# B&R Automation Studio project EFI (part 13)

#### Documentation.txt - Release Axis Ctrl Logic
```
 **************************************************************************************************
 * COPYRIGHT - B&R Spain
 **************************************************************************************************
 * Program: AxisCtrl
 * File: Documentation.txt
 * Author: B&R Spain
 * Created: September 19, 2013
 * Modified: April 28, 2017
 **************************************************************************************************
 * Implementation of program AxisCtrl
 **************************************************************************************************
 * V 0.03.4
 **************************************************************************************************

 * Requirements
 **************************************************************************************************

 - ACP10 version must be equal or higher than V2.26.0 because before that version the ACP10_MC FBK
   errors were not read by the MC_ReadAxisError FBK and therefore a lot of diagnostic information
   would be lost in case a previous version would be used.

 * Configuration
 **************************************************************************************************

 - The file References.st must be updated to allow the program to control the desired axis. This is
   the only part of the program that needs to be modified if the functionality does not need to be
   changed.

 - It must be noted that the name of the control variable is not used inside the program to avoid
   requiring a Find & Replace. The control variable just needs to be specified in the references.st
   file.

 * Functionality
 **************************************************************************************************

 - The funtionality is very similar to the SingleAx or Basic one. It basically has some expansions
   to allow higher flexibility. The interface is quite easy to use. Furthermore, there are some
   differences compared to the SingleAx and Basic programs, which are described in the following
   chapter.

 - The control structure is divided in three parts; the commands, the parameters and the status.

 - In addition to the PLCopen state, the control structure provides useful status information like
   the PowerOn, the HomeOk and the InPosition that reflects if the axis is switched on, if it is
   properly homed and if the last commanded discrete movement has reached the target, respectively.
   The status structure provides information about the ACOPOS digital inputs as well.

 * Main differences in behaviour compared to the SingleAx and Basic
 **************************************************************************************************

 - In this program, all the valid PLCopen transitions are possible. E.g. While a MoveAbsolute is
   performed (DiscreteMotion), a MoveVelocity can be started (ContinuousMotion). This includes as
   well performing a MoveAbsolute to a new target while a MoveAbsolute is in process. Not all the
   combinations were possible in the SingleAx and Basic programs.

 - Instead of a Stop, this program provides a Halt and a QuickStop.
   - The Halt allows Discrete, Continuous and synchronized movements to be halted (Discrete motion
     where the speed is decreased until it becomes zero). This allows a higher flexibility since
	 the Halt itself can be aborted by another movement or even a new Halt with other parameters.
	 This would be not possible if a Stop would be used.
   - The QuickStop performs a stop with the limit deceleration (Axis init table). The QuickStop can
     be thought of a "panic" stop. It has higher priority than any other command except switching
	 off the drive. If the QuickStop is set, no movement will be allowed to start. In case any un-
	 expected error occurrs, the QuickStop should be used to stop the motion.

 - The Quickstop and the Power must be reset by the application. This program will never reset them.

 - In this program, only the real axis errors (i.e. the ones that bring the axis to ErrorStop in
   the PLCopen state diagram. E.g. encoder fault) cause the axis to stop. If other errors (e.g.
   warnings or ACP10_MC errors (29xxx) occurr), the axis remains in its last state and can be ope-
   rated as normal. Therefore, the errors can be read (Acknowledged) while the axis is in motion.
   However, every error which is reported should be considered by the application and if necessary,
   command a QuikStop.

 - As the PLCopen state diagram states, the Reset command can be used to leave the ErrorStop state
   directly with no need to acknowledge the errors one by one. To mantain backwards compatibility,
   if all errors are acknowledged by the ErrorAcknowledge command, the axis leaves the ErrorStop
   state as well.

 - In this program, the homming mode cannot be specified by the application. Instead, there are
   three kind of home commands, which is enough for almost all applications.
   - The HomeDirect, which assigns a value to the actual position. This command can be used either
     in standstill or in disabled state.
   - The HomeAbsEncoder, which takes into account the absolute encoder to calculate the position.
     This command can be used either in standstill or in disabled state. To allow this functionality
	 a permanent variable must be linked, where the program will store the necessary data for it.
   - The Home, which performs a home in the way it is defined in the axis parameter table. this is
     the only home command that can cause the axis to move.

 - In this program, there are two kind of Jog commands; a continuous and an incremental one.

 - By default, if a command is set, which is not allowed at the time, the program returns an error.
   This behaviour can be changed by commenting the corresponding part of the program.

 - By default, if two or more incoherent commands are set at the same time, the axis ignores and
   resets all the commands (exept the QuickStop and the Power). This behaviour can be changed by
   commenting the corresponding part of the program.

 - This program has been designed to avoid all the known bugs from the SingleAx and Basic programs.

 - This program also fixes some ACP10 flaws. E.g. this program does not allow a periodic axis to be
   moved if it is not properly homed. This is not prevented by ACP10, and it might lead to very dan-
   gerous movements where the axis could collide against other machine parts.

 - There is a PLCopen state supervisor that makes sure that even if the axis is commanded by an ex-
   ternal source (e.g. the Test Window), it will always be possible to operate it from the program
   side (of course not while the Test is opened in Exclusive mode, but will work after it is closed).
   However, it is recommended not to move the axis from the Test Window, since the changes that it
   does are not monitored by PLCopen FBs. Moving the axis from the test window can cause the next
   movements to use speeds and accelerations other than the ones programmed.

 - The way the program gets access to the axes (ncaccess) makes sure that the program can be trans-
   fered in any mode (overload, copy or one cycle) and the program will still be able to manage the
   axis. No warm restart will be required, even after the first transfer.

 * Modifications: Recommended way to modify the program
 **************************************************************************************************

  In order to implement changes that require the use of a state machine, it is not always
  necessary to expand/modify the main sequence (AxisState state machine). Consider the possibility
  to use a new state machine specifically for that functionality. It will be much easier to
  implement and it will actually make more sense if it is not part of the main sequence. For
  instance, this would be the case of a manual brake operation, where the main sequence step does
  not need to be considered if the higher level application requires to set or release the brake.

  Depending on the changes to implement there are different strategies to follow:

  - If the program must be expanded but the main sequence is not going to be changed, for example
    in case the ActualTorque must be read, the program can be expanded just by doing as follows:

    1)  Modify the control structure AxisCtrl_typ or any derivative, and all necessary substructures.
    2)  Declare all needed FBKs instances and temporary variables.
    3)  Implement the FBK parameterization and call in the corresponding FBK call section in the
        AxisCtrl.st file.
    4)  Update the status values of the control structure in the last part of the AxisCtrl.st file.

  - In order to modify the main sequence in an appropiate way, next steps must be followed:

    1)  Modify the control structure AxisCtrl_typ or any derivative, and all necessary
        substructures.
    2)  Declare all needed FBKs instances and any temporary variable (AxisCtrl.var file). In case
        of movement FBKS, declare two instances ended in _0 and _1 to allow two consecutive motion
        commands of the same type.
    3)  Expand the AxisState_typ enumeration (AxisCtrl.typ file) to include the new required steps.
        In case of motion states, declare two states ended in _0 and _1 to allow two consecutive
        motion commands of the same type.
    4)  Define all the new necessary actions in the Commands.st file. In case of movement actions,
        declare two actions ended in _0 and _1 to allow two consecutive motion commands of the
        same type.
    5)  Add code to reset all the new commands in the ResetMotionCommands action (Commands.st).
    6)  Add code to reset all the new FBKs in the ResetExecutes action (Commands.st).
    7)  Implement the new steps in the CASE of the AxisCtrl.st file by following the same style
        used in the other steps.
    8)  Implement the FBK parameterization and call in the corresponding FBK call section in the
        AxisCtrl.st file.
    9)  Add the newly created steps in the CASE of the StateSupervisor.st considering in which
        PLCopen state the axis must be for each step, in order to detect any anomaly in the axis
        state.
    10) Add the possibility to perform the command (e.g. Move.CyclicPosition) wherever it should
        be possible (i.e. in every step of the CASE where it should be possible to do so) in the
	    AxisCtrl.st file. Keep the same style which is used in the other steps.
    11) In order to detect if any command is commanded when it connot be, add the corresponding
        code in the COMMAND INCOHERENCE CHECK section in the AxisCtrl.st file.
    12) In order to detect if two incoherent commands are commanded at the same time, add the
        corresponding code in the INVALID COMMAND ABORTION section in the AxisCtrl.st file.
    13) Update the status values of the control structure in the last part of the AxisCtrl.st file
        if necessary.
    14) Document all the important behavioural changes of the task in the Documentatioin.txt file.

 **************************************************************************************************
 * Revision History
 **************************************************************************************************
 * V0.03.4  2017-04-28
 * (change) Virtual axes exhibit now the same bahviour as real axes (PowerOn status corresponds to
 * the Power command and PLCopenState.Disabled and PLCopenState.Standstill status are consistent
 * to the Power command).
 * (change) The Power command is not set to TRUE by the program any more, because there is no need.
 * (bug fix) PowerOn status was set too early and that could incorrectly lead to error 29207
 * (bug fix) Some AR version (e.g. F4.03) do not copy the pointer's address when transferring in
 * copy mode. The program can work fine now with those AR versions as well.
 **************************************************************************************************
 * V0.03.3  2016-07-26
 * (Bug fix) The battery-backed (EBI) encoder errors were reset in more cases than strictly needed
 **************************************************************************************************
 * V0.03.2  2016-07-26
 * (new) Battery-backed (EBI) encoder errors can be directly acknowledged via the ErrorAcknowledge
 * command, for example during the first startup or after the encoder cable has been disconnected.
 * Internally, the task writes the ENCOD_COMMAND ParID to reset the econder error when necessary.
 * It must be noted that it is not possible to recover from a battery-backed (EBI) encoder error
 * via the Reset command. Only the ErrorAcknowledge command can recover the situation.
 * (new) If a battery-backed (EBI) encoder error is detected, the permanent memory that is used by
 * the mcHOME_RESTORE_POS is set to be invalid, because the absolute position could be wrong.
 * (Bug fix) Error message for MC_BR_AutControl was not correct
 **************************************************************************************************
 * V0.03.1  2016-02-17
 * (bug fix) If the axis lost the HomeOK due to an encoder error, the ActualPosition did not change
 * to NaN and the workaround introduced in V0.03.0 for the APC10 flaw was not preventing the axis
 * to move after an encoder error.
 * (bug fix) If the axis is not synchronized anymore due to an external abortion (e.g. because it
 * was stopped from the Test Window), the InGear and InSynch flag was not reset.
 * (change) Now the CommandAborted output from the different FBs is used to detect sooner if an
 * external agent (e.g the Test Window) is commanding other movements.
 * (change) If the program was transfered in overload mode while the axis state was not Standstill
 * or Disabled, the MC_BR_InitEndlessPosition was filling the error FIFO. Now it waits until it
 * can be executed and the InitDone remains FALSE until then.
 **************************************************************************************************
 * V0.03.0  2016-02-10
 * (change) If the axis is not properly referenced (HomeOK = FALSE), the ActualPosition shows Not
 * a Number (NaN) in order to avoid confusions.
 * (change) Error 50001 has been replaced by error 29207, which provides a more precise description
 * with detailed information about the FB which is responsible for it, making it easier to diagnose
 * application problems.
 * (new) If the axis is not properly referenced (HomeOK = FALSE), the axis is not allowed to
 * move by the application and error 29205 is reported. This is done because there is an ACP10 flaw
 * that allows rotary axes to move even if they are not homed and that could lead to dangerous
 * movements that might end colliding against some other machine part.
 * (new) The Status member ErrorSource has been added so that it is possible to know if the actual
 * error message has been reported by ACP10, by PLCopen or by the Task itself.
 * (new) The MC_BR_InitAutData has been added in the AutCtrl program to be able update the automat
 * parameters in a faster way after a second StartAutomat command.
 **************************************************************************************************
 * V0.02.9  2015-12-24
 * (new) The member PowerOn has been added to the Status structure so that it is possible to know
 * if power is supplied to the axis by just looking at it.
 **************************************************************************************************
 * V0.02.8  2015-05-06
 * (change) If the axis to control is a virtual axis, the Power command is automatically set to
 * TRUE by the program so that it will not cause PLCopen conflicts. This is because virtual axes
 * cannot be in Disabled state and the state supervisor would try to switch the axis off repeatedly
 * until the Power command would be set to TRUE.
 **************************************************************************************************
 * V0.02.7  2014-02-18
 * (new) There is a new sample (CamCtrl) to handle a cam profile coupling. Note that the Move.CamIn
 * command can only be used while the axis is not in SynchronizedMotion, so that to CamIn a second
 * time, first a CamOut or another aborting command must be commanded.
 * (new) There is a new sample (AutCtrl) to handle a cam profile automat coupling. Note that the
 * Move.StartAutomat command can be used while the axis is not in SynchronizedMotion to start the
 * automat, but can be commanded again to update the automat parameters during runtime.
 * (change) The GearOut did not work correctly.
 **************************************************************************************************
 * V0.02.6  2013-12-30
 * (change) The state supervisor has been changed so that if an exception is found, it takes into
 * account the actual state for every cicle, without waiting for any timeout. This was necessary
 * when the CNC/robotics was used, because the axis was changed to synchronized motion and back to
 * standstill by the CNC and then it was not possible to perform any movement before the timeout
 * expired.
 **************************************************************************************************
 * V0.02.5  2013-10-17
 * (new) There is a new sample (GearCtrl) to handle a gear coupling.
 * (change) The way to handle the FBK calls has changed to let the user know when the master axis
 * is not correct.
 **************************************************************************************************
 * V0.02.4  2013-09-30
 * (new) First internally released version.
 **************************************************************************************************
```

#### AxisCtrl.typ - Local data types
```iecst
(********************************************************************
 * COPYRIGHT - B&R Spain
 ********************************************************************
 * Program: AxisCtrl
 * File: AxisCtrl.typ
 * Author: B&R Spain
 * Created: September 19, 2013
 ********************************************************************
 * Local data types of program AxisCtrl
 ********************************************************************)

TYPE
	AxisState_typ :
		(
		AX_STATE_DISABLED := 0,
		AX_STATE_HOMING_NO_POWER := 1,
		AX_STATE_SWITCHING_OFF := 2,
		AX_STATE_STANDSTILL := 10,
		AX_STATE_SWITCHING_ON := 11,
		AX_STATE_STOPPING := 12,
		AX_STATE_HOMING := 13,
		AX_STATE_MOVING_ABSOLUTE_0 := 20,
		AX_STATE_MOVING_ABSOLUTE_1 := 21,
		AX_STATE_MOVING_ADDITIVE_0 := 22,
		AX_STATE_MOVING_ADDITIVE_1 := 23,
		AX_STATE_MOVING_VELOCITY_0 := 24,
		AX_STATE_MOVING_VELOCITY_1 := 25,
		AX_STATE_MOVING_GEAR_0 := 40,
		AX_STATE_MOVING_GEAR_1 := 41,
		AX_STATE_HALTING_0 := 26,
		AX_STATE_HALTING_1 := 27,
		AX_STATE_JOGGING_POS := 30,
		AX_STATE_JOGGING_NEG := 31,
		AX_STATE_JOGGING_SS_POS := 32,
		AX_STATE_JOGGING_SS_NEG := 33,
		AX_STATE_JOG_SS_HALTED := 34,
		AX_STATE_HALTING_JOG := 35,
		AX_STATE_UNKNOWN := 200,
		AX_STATE_UK_DISABLED := 201,
		AX_STATE_UK_STANDSTILL := 202,
		AX_STATE_UK_HOMING := 203,
		AX_STATE_UK_DISCRETE_MOTION := 204,
		AX_STATE_UK_CONTINUOUS_MOTION := 205,
		AX_STATE_UK_SYNCHRONIZED_MOTION := 206,
		AX_STATE_UK_STOPPING := 207,
		AX_STATE_UK_ERROR_STOP := 208
		);
	AxisErrorState_typ :
		(
		AX_ERR_STATE_WAIT := 100, (*constant for the waiting error step*)
		AX_ERR_STATE_APP_ERROR := 101, (*constant for the application error step*)
		AX_ERR_STATE_AXIS_ERROR := 102, (*constant for the axis error step*)
		AX_ERR_STATE_ENCODER_RESET := 103 (*constant for the step where the encoder error is reset*)
		);
END_TYPE
```

- Program Logical/ExtPack/_Motion/AxisCtrl/AxisCtrl_v2/InitAxisControl (IEC) - Init Axis Control Index (no source held here)

### AxisCtrlGen.var - Global Axis Vars
```iecst
VAR
	gIndexAxisCtrl : INT := 1; (* Initialize Index*)
END_VAR
```

### Icla.typ
```iecst
(*********************************************************************************
 * Copyright: Bernecker + Rainer
 * Author:    gimeneza
 * Created:   June 15, 2017/4:14 PM
 *********************************************************************************)

TYPE
	stIcla_Error : 	STRUCT
		Jog : BOOL;
		Communication : BOOL;
		ErrorNumber : UINT;
	END_STRUCT;
	stIcla_Jog : 	STRUCT
		VeloSlow : UINT := 300; (*Rev/min Limited from 300 to 5000. 300 is the default value in Icla*)
		VeloFast : UINT := 1000; (*Rev/min Limited from 300 to 5000. 1000 is the default value in Icla*)
	END_STRUCT;
	stIcla_MoveAbsolute : 	STRUCT
		Position : DINT;
		Velocity : UINT;
	END_STRUCT;
	stIcla_Homing : 	STRUCT
		Position : DINT;
		Mode : USINT;
	END_STRUCT;
	stIcla_Commands : 	STRUCT
		Enable : BOOL;
		Home : BOOL; (*EDGE to Home the drive. Reseted when starting Home process*)
		MoveAbsolute : BOOL;
		JogForward : BOOL;
		JogBackward : BOOL;
		JogFastSpeed : BOOL;
		Stop : BOOL; (*EDGE*)
		Reset : BOOL; (*EDGE*)
	END_STRUCT;
	stIcla_RegistersValueArray : 	STRUCT
		data0 : USINT; (*data of the register. USINT*)
		data1 : USINT; (*data of the register. USINT*)
		data2 : USINT; (*data of the register. USINT*)
		data3 : USINT; (*data of the register. USINT*)
	END_STRUCT;
	stIcla_RegistersValue : 	STRUCT
		usiValue : USINT; (*Value of data0, just for USINT data. 8 bits*)
		uiValue : UINT; (*Value of data0 & data1, just for UINT data. 16bits*)
		xDataOK : BOOL; (*Data in values is correct*)
		xBusy : BOOL; (*The registers are beeing read*)
		rawData : stIcla_RegistersValueArray; (*raw USINT data array from communication function*)
	END_STRUCT;
	stIcla_Register : 	STRUCT
		index : USINT := 1; (*Index of the register to read. 1:2 by default is Firmware version*)
		subindex : USINT := 2; (*Subindex of the register to read. 1:2 by default is Firmware version*)
	END_STRUCT;
	stIcla_WriteRegister : 	STRUCT
		WriteOrder : BOOL;
		TotalBytes : USINT := 2; (*Quantity of bytes to send Just 2 and 4 are valid values*)
		data : stIcla_RegistersValueArray := (0); (*Bytes of Data to send*)
		writeRegister : stIcla_Register; (*Register to write the data in the Icla while the comms are in idle*)
	END_STRUCT;
	stIcla_Parameters : 	STRUCT
		Home : stIcla_Homing;
		MoveAbsolute : stIcla_MoveAbsolute;
		Jog : stIcla_Jog;
		Node : USINT := 255; (*255 is the maximum value of USINT. It means the node is still not configured *)
		Network : STRING[7]; (*The Position of the network*)
		iAcceleration : UINT := 2500; (*Acceleration of the Icla revolutions min^-1/sec. Limited to 1000 and 10000 by the Icla itself. 2500 is the default value*)
		xAutoresetComms : BOOL; (*Send NMT message if not communicating to restore communication with an Icla*)
		readRegister : stIcla_Register; (*Read registers from the Icla while the comms are in idle*)
		writeRegister : stIcla_WriteRegister; (*Read registers from the Icla while the comms are in idle*)
	END_STRUCT;
	stIcla_Status : 	STRUCT
		xModuleOK : BOOL;
		xIsHoming : BOOL;
		xReferenced : BOOL;
		xInError : BOOL;
		xInPosition : BOOL; (*Edge*)
		iActualPosition : DINT;
		iActualVelocity : INT;
		iDriveStatus : UINT;
		Error : stIcla_Error;
		Info : STRING[80];
		IclaStatus : stepAXISILE_enum;
		IclaSDOStep : stepCOMSILE_enum;
		readRegister : stIcla_RegistersValue;
		writeRegisterOK : BOOL;
	END_STRUCT;
	stIcla : 	STRUCT
		Command : stIcla_Commands;
		Parameter : stIcla_Parameters;
		Status : stIcla_Status;
	END_STRUCT;
	TPDO4_typ : 	STRUCT
		modeStat : USINT;
		driveStat : UINT;
		Act8 : SINT;
		Act32 : DINT;
	END_STRUCT;
	RPDO4_typ : 	STRUCT
		driveCtrl : USINT;
		modeCtrl : USINT;
		ModuleOK : BOOL;
		Ref16 : INT;
		Ref32 : DINT;
	END_STRUCT;
	IclaNetData_typ : 	STRUCT
		RPDO4 : RPDO4_typ;
		TPDO4 : TPDO4_typ;
		xModuleOK : BOOL;
	END_STRUCT;
	stepAXISILE_enum :
		(
		AXISILE_INIT,
		AXISILE_WAIT_READY_TO_SWITCH_ON,
		AXISILE_DOWNLOAD,
		AXISILE_CONFIRM,
		AXISILE_ACKN,
		AXISILE_UNLOCK,
		AXISILE_WAIT,
		AXISILE_POWER,
		AXISILE_HOMING,
		AXISILE_READY,
		AXISILE_JOG,
		AXISILE_MOVE_ABSOLUTE,
		AXISILE_ERROR
		);
	stepCOMSILE_enum :
		(
		COMSILE_IDLE,
		COMSILE_ACCELERATION,
		COMSILE_JOG_PAUSE,
		COMSILE_JOG_TRANSFER_SLOW,
		COMSILE_JOG_TRANSFER_FAST,
		COMSILE_READ_SPEED,
		COMSILE_ERROR
		);
END_TYPE
```

### Program Logical/ExtPack/_Motion/IclaCtrl/IclaCtrl_v4/IclaCtrl (IEC)

#### ResetComms.st
```iecst
ACTION ResetComms:

	CanGetState.enable := TRUE;
	CanGetState.node := Icla.Parameter.Node;
	CanGetState.pDevice := ADR(Icla.Parameter.Network);
	CanGetState();

	iReasonNotComms.0 := CanGetState.state = coPREOPERATIONAL;
	iReasonNotComms.1 := CanGetState.state = coUNKNOWN;
	iReasonNotComms.2 := CanGetState.state = coNOTAVAIL;
	iReasonNotComms.3 := NOT Icla.Status.xModuleOK;

	tonNotComms.IN := iReasonNotComms > 0;
	tonNotComms.PT := t#3s;
	tonNotComms();

	xChangedResetCommsState := CanResetState_copy <> CanResetState;
	CanResetState_copy := CanResetState;

	CASE CanResetState OF

		COCOMSR_UNDEFINED,
		COCOMSR_COMMUNICATING:

			iTimesTryToReset := 0;

			//If time in error, define an error comms
			IF tonNotComms.Q THEN
				CanResetState := COCOMSR_COMMSERROR;
			END_IF

		COCOMSR_COMMSERROR:

			//Start the resetting process
			IF Icla.Command.Reset AND Icla.Parameter.xAutoresetComms THEN
				CanResetState := COCOMSR_RESETTING;
			END_IF

			//Communication has returned to work
			IF CanGetState.state = coOPERATIONAL THEN
				CanResetState := COCOMSR_COMMUNICATING;
			END_IF

		COCOMSR_RESETTING:

			CANopenReset.enable := TRUE;
			CANopenReset.node := Icla.Parameter.Node;
			CANopenReset.pDevice := ADR(Icla.Parameter.Network);
			CANopenReset.state := coRESET_NODE;
			CANopenReset();

			IF CANopenReset.status = ERR_OK THEN
				lastCanOpenResetError := CANopenReset.error;
				CANopenReset(enable := FALSE);
				CanResetState := COCOMSR_WAITINGTOBERESETTED;
			END_IF

			tonCommsErrorResetting.IN := NOT xChangedResetCommsState;
			tonCommsErrorResetting.PT := t#10s;
			tonCommsErrorResetting();

			IF tonCommsErrorResetting.Q THEN
				lastResetingState := CanGetState.state;
				lastFbResetStatus := CANopenReset.status;
				tonCommsErrorResetting(IN:=FALSE);
				CANopenReset(enable:=FALSE);
				CanResetState := COCOMSR_RESETTING_ERROR;
			END_IF

		COCOMSR_WAITINGTOBERESETTED:

			//Communication has returned to work
			IF CanGetState.state = coOPERATIONAL THEN
				CanResetState := COCOMSR_COMMUNICATING;
			END_IF

			tonCommsErrorResetting.IN := NOT xChangedResetCommsState;
			tonCommsErrorResetting.PT := t#4s;
			tonCommsErrorResetting();

			IF tonCommsErrorResetting.Q THEN
				lastResetingState := CanGetState.state;
				lastFbResetStatus := CANopenReset.status;
				tonCommsErrorResetting(IN:=FALSE);
				CanResetState := COCOMSR_RESETTING_ERROR;
			END_IF

		COCOMSR_RESETTING_ERROR:

			//After an error, wait to try again
			tonCommsErrorResetting.IN := NOT xChangedResetCommsState;
			tonCommsErrorResetting.PT := t#500ms;
			tonCommsErrorResetting();

			IF tonCommsErrorResetting.Q  AND iTimesTryToReset < 6 THEN
				iTimesTryToReset := iTimesTryToReset + 1;
				CanResetState := COCOMSR_RESETTING;
			ELSIF tonCommsErrorResetting.Q THEN
				CanResetState := COCOMSR_COMMSERROR;
			END_IF

	END_CASE;

END_ACTION
```

### Program Logical/ExtPack/_Motion/IclaCtrl/IclaSim/IclaSim_v1/InitIclaSim (IEC)

#### Main.st
```iecst
PROGRAM _CYCLIC

	iIclaSimIndex := 1;

END_PROGRAM
```

### Program Logical/ExtPack/_Motion/InverterCtrl/InverterCtrl_v1/InverterCtrl (IEC, version 1.01.0) - Controls an P66/P76 ACOPOSinverter

#### InverterCtrl.st - Implementation code
```iecst
(********************************************************************
 * COPYRIGHT -- Bernecker + Rainer
 ********************************************************************
 * Program: I66Ctrl
 * File: I66Ctrl.st
 * Author: tresensa
 * Created: May 09, 2014
 ********************************************************************
 * Implementation of program InvCtrl
 ********************************************************************)

PROGRAM _INIT

	ErrorTable;	(* Writes the error table *)

	ErrorTableACS380;	(* Writes the error table *)

	ErrMessage_FUB.Enable	:= TRUE;
	ErrMessage_FUB.ErrList	:= Error;

	RTInfo_0(enable:=TRUE); (* Get cycle time *)
	SimCycleTime := UDINT_TO_REAL(RTInfo_0.cycle_time) / 1000000; (* Conversion to seconds *)

END_PROGRAM

PROGRAM _CYCLIC

	dataInv ACCESS ADR (gAxisInverter[iIndexInverter]);

	CASE dataInv.Parameters.CommsType OF
		COMMS_POWERLINK:
			CASE dataInv.Parameters.Type OF
				INV_BR:
					ioMap ACCESS ADR (gInverterSignalsPowerLink[iIndexInverter]);
				INV_ABB:
					ioMap ACCESS ADR (gInverterSignalsPowerLinkABB[iIndexInverter]);
			END_CASE;

		COMMS_CANOPEN: 		ioMap ACCESS ADR (gInverterSignalsCanOpen[iIndexInverter]);

		ELSE
			//If comms type is not configured, go to next inverter
			//Prepare the index for the next Inverter
			dataInv.Status.ErrorComms := TRUE;
			iIndexInverter := iIndexInverter + 1;
			RETURN;
	END_CASE

	ResetComms;

	GenInverterCtrl;

	//Prepare the index for the next Inverter
	iIndexInverter := iIndexInverter + 1;

END_PROGRAM
```

#### GenInvCtrl.st - Implementation code
```iecst
ACTION GenInverterCtrl:

(********************************************************************************
*********************************************************************************

	INFORMATION OF POWERLINK DEVICES

	EXAMPLE Program for Handling of a P74 Inverter
	Task: I74Ctrl Program

	<|> Structure to handle the axis:

		Name								Format		Type		Description
		---------------------------------------------------------------------------------------------------------
		dataInv.Orders.PowerOn				| BOOL		| Command	| Switches the power on
		dataInv.Commands.MovePositive		| BOOL		| Command	| Starts a movement in the positive direction
		dataInv.Commands.MoveNegative		| BOOL		| Command	| Starts a movement in the negative direction
		dataInv.Commands.Stop				| BOOL		| Command	| Stops the axis
		dataInv.Commands.Reset				| BOOL		| Command	| Acknowledges and quits all errors
		dataInv.Parameters.Velocity		| INT		| Parameter	| Set speed
		dataInv.Parameters.AccelerationTime			| UINT		| Parameter	| Set acceleration time
		dataInv.Parameters.DecelerationTime			| UINT		| Parameter	| Set deceleration time
		dataInv.Status.ActVelocity			| INT		| Status	| Actual speed
		dataInv.Status.ActCurrent			| UINT		| Status	| Actual current
		dataInv.Status.ActTorque			| UINT		| Status	| Actual torque
		dataInv.DigitalInput		| BOOL[8]	| Status	| Digital Inputs of the inverter [0...7]
		dataInv.DigitalOutput		| BOOL[3]	| Status	| Digital Outputs of the inverter [0...2]
		dataInv.AnalogInput			| INT[3]	| Status	| Analog Inputs of the inverter [0...2]
		dataInv.AnalogOutput		| UINT		| Status	| Analog Output of the inverter
		dataInv.Status.ErrorID				| UINT		| Status	| Error number
		dataInv.Status.ErrorText			| STRING[9]	| Status	| Error description
		dataInv.Status.StatusDisabled		| BOOL		| Status	| The inverter is switched off
		dataInv.Status.StatusReady			| BOOL		| Status	| The inverter is ready to perform a movement
		dataInv.Status.StatusOperation		| BOOL		| Status	| The motor is powered
		dataInv.Status.StatusErrorStop		| BOOL		| Status	| The inverter has some error

	<|> Variables that need to be mapped in the IO Mapping of the Inverter:

		IO Point		Format		Local Variable			Addtitional
		----------------------------------------------------------------
		ModuleOk		| BOOL		| ioMap.In.ModuleOk		| Compulsory
		ETAD_Input		| UINT		| ioMap.In.StatusWord		| Compulsory
		RFRD_Input		| INT		| ioMap.In.ActualSpeed		| Optional
		LCR_Input		| UINT		| ioMap.In.ActualCurrent	| Optional
		OTRN_Input		| UINT		| ioMap.In.ActualTorque	| Optional
		LFT_Input		| INT		| ioMap.In.ErrorID			| Optional
		CMDD_Output		| UINT		| ioMap.Out.ControlWord		| Compulsory
		LFRD_Output		| INT		| ioMap.In.SetSpeed		| Compulsory
		IL1R_Input_DI1	| BOOL		| ioMap.In.DigitalInput[0]	| Optional
		IL1R_Input_DI2	| BOOL		| ioMap.In.DigitalInput[1]	| Optional
		IL1R_Input_DI3	| BOOL		| ioMap.In.DigitalInput[2]	| Optional
		IL1R_Input_DI4	| BOOL		| ioMap.In.DigitalInput[3]	| Optional
		IL1R_Input_DI5	| BOOL		| ioMap.In.DigitalInput[4]	| Optional
		IL1R_Input_DI6	| BOOL		| ioMap.In.DigitalInput[5]	| Optional
		IL1R_Input_DAI1	| BOOL		| ioMap.In.DigitalInput[6]	| Optional
		IL1R_Input_DAI2	| BOOL		| ioMap.In.DigitalInput[7]	| Optional
		OL1R_Output_R1	| BOOL		| ioMap.In.DigitalOutput[0]| Optional
		OL1R_Output_R2	| BOOL		| ioMap.In.DigitalOutput[1]| Optional
		OL1R_Output_RDQ1| BOOL		| ioMap.In.DigitalOutput[2]| Optional
		AI1R_Input		| INT		| ioMap.In.AnalogInput[0]	| Optional
		AI2R_Input		| INT		| ioMap.In.AnalogInput[1]	| Optional
		AI3R_Input		| INT		| ioMap.In.AnalogInput[2]	| Optional
		AO1R_Output		| UINT		| ioMap.In.AnalogOutput	| Optional

*********************************************************************************)

(********************************************************************************
*********************************************************************************

	INFORMATION OF CANOPEN DEVICES

	EXAMPLE Program for Handling of a X64 Inverter
	Task: I66Ctrl Program
	(c) 2010 by B&R-ES

	<|> Structure to handle the axis:

		Name								Format		Type		Description
		---------------------------------------------------------------------------------------------------------
		gAxisInverter01.PowerOn				| BOOL		| Command	| Switches the power on
		gAxisInverter01.MovePositive		| BOOL		| Command	| Starts a movement in the positive direction
		gAxisInverter01.MoveNegative		| BOOL		| Command	| Starts a movement in the negative direction
		gAxisInverter01.Stop				| BOOL		| Command	| Stops the axis as configured in FUN->STC->STT (Default: RMP)
		gAxisInverter01.Reset				| BOOL		| Command	| Acknowledges and quits all errors
		gAxisInverter01.ParaVelocity		| INT		| Parameter	| Set speed [rpm]
		gAxisInverter01.ParaAccTime			| UINT		| Parameter	| Set acceleration time [s]
		gAxisInverter01.ParaDecTime			| UINT		| Parameter	| Set deceleration time [s]
		gAxisInverter01.ActVelocity			| INT		| Status	| Actual speed [rpm]
		gAxisInverter01.ActCurrent			| REAL		| Status	| Actual current [A]
		gAxisInverter01.ActTorque			| REAL		| Status	| Actual torque [Nm]
		gAxisInverter01.ErrorID				| UINT		| Status	| Error number
		gAxisInverter01.ErrorText			| STRING[9]	| Status	| Error description
		gAxisInverter01.StatusDisabled		| BOOL		| Status	| The inverter is switched off
		gAxisInverter01.StatusReady			| BOOL		| Status	| The inverter is ready to perform a movement
		gAxisInverter01.StatusOperation		| BOOL		| Status	| The motor is powered
		gAxisInverter01.StatusErrorStop		| BOOL		| Status	| The inverter has some error
		gAxisInverter01.DigitalInput[0..5]	| BOOL		| Input		| Digital inputs
		gAxisInverter01.DigitalOutput		| BOOL		| Output	| Digital Output
		gAxisInverter01.AnalogInput[0..2]	| INT		| Input		| Analog inputs
		gAxisInverter01.DigitalOutput		| UINT		| Output	| Analog Output

	<|> Variables that need to be mapped in the IO Mapping of the Inverter:

		IO Point		Format		Local Variable			Addtitional
		----------------------------------------------------------------
		ModuleOk		| BOOL		| ioMap.ModuleOk		| Compulsory
		ETAD_Input		| UINT		| ioMap.StatusWord		| Compulsory
		RFRD_Input		| INT		| ioMap.ActualSpeed		| Compulsory
		LCR_Input		| UINT		| ioMap.ActualCurrent	| Optional
		LFT_Input		| INT		| ioMap.ErrorID			| Optional
		CMDD_Output		| UINT		| ioMap.ControlWord		| Compulsory
		LFRD_Output		| INT		| ioMap.SetSpeed		| Compulsory

	EXAMPLE Program FOR Handling OF a ABB ACS380	Task: ACS380 Program

		<|> Structure TO handle the axis:

		Name								Format		Type		Description
		---------------------------------------------------------------------------------------------------------
		gAxisInverter01.PowerOn				| BOOL		| Command	| Switches the power on
		gAxisInverter01.MovePositive		| BOOL		| Command	| Starts a movement in the positive direction
		gAxisInverter01.MoveNegative		| BOOL		| Command	| Starts a movement in the negative direction
		gAxisInverter01.Stop				| BOOL		| Command	| Stops the axis
		gAxisInverter01.Reset				| BOOL		| Command	| Acknowledges AND quits all errors
		gAxisInverter01.ControlMode			| UINT		| Parameter	| Chose control mode. 0 = VECTOR // 1 = SCALAR
		gAxisInverter01.ParaVelocity		| INT		| Parameter	| Set speed
		gAxisInverter01.ParaAccTime			| UINT		| Parameter	| Set acceleration time
		gAxisInverter01.ParaDecTime			| UINT		| Parameter	| Set deceleration time
		gAxisInverter01.ActVelocity			| INT		| Status	| Actual speed
		gAxisInverter01.ActCurrent			| UINT		| Status	| Actual current
		gAxisInverter01.ErrorID				| UINT		| Status	| Error number
		gAxisInverter01.ErrorText			| STRING[9]	| Status	| Error description
		gAxisInverter01.StatusDisabled		| BOOL		| Status	| The inverter is switched off
		gAxisInverter01.StatusReady			| BOOL		| Status	| The inverter is ready TO perform a movement
		gAxisInverter01.StatusOperation		| BOOL		| Status	| The motor is powered
		gAxisInverter01.StatusErrorStop		| BOOL		| Status	| The inverter has some error

		<|> Variables that need TO be mapped in the IO Mapping OF the Inverter:

		IO Point									Format		Local Variable			Addtitional
		-------------------------------------------------------------------------------------------------------------
		ModuleOk									| BOOL		| ioMap.ModuleOk		| Compulsory
		ABBSW_I2104									| UINT		| ioMap.StatusWord		| Compulsory
		ABBAct1_I2104								| INT		| ioMap.ActualSpeed		| Optional
		CurrentActualValue_I6078					| INT		| ioMap.ActualCurrent	| Optional
		ErrorCode_I603F								| UINT		| ioMap.ErrorID			| Optional
		ABBCW_I2101Out								| UINT		| ioMap.ControlWord		| Compulsory
		ABBRef1_I21012Out							| INT		| ioMap.SetSpeed		| Compulsory
		ABBRef1_I21013Out							| INT		| ioMap.SetFrequency	| Compulsory
		_9904_Motor_control_mode_I4060_S08Out		| UINT		| ioMap.ControlMode		| Optional
		_5004_FBA_A_ref1_type_I4032_S04Out			| UINT		| ioMap.SpeedUnit		| Compulsory
		_2312_Acceleration_time_1_I4017_S0COut		| DUINT		| ioMap.AccTimeVector	| Compulsory
		_2313_Deceleration_time_1_I4017_S0DOut		| DUINT		| ioMap.DecTimeVector	| Compulsory
		_2872_Freq_acceleration_time_1_I401C_S48Out	| DUINT		| ioMap.AccTimeScalar	| Compulsory
		_2873_Freq_deceleration_time_1_I401C_S49Out	| DUINT		| ioMap.DecTimeScalar	| Compulsory

		*********************************************************************************)

	(* Module Information *)
	PL_device := dataInv.Parameters.Hardware.PowerLinkInterface; 	// (* Powerlink interface *)  originally 'SL1.IF3';
	HW_node := dataInv.Parameters.Hardware.Node; 					// (* Powerlink station (node number of the inverter) *) originally 2;

(********************************************************************
	Parameter Transfer: ACC, DEC (valid for P66)
*********************************************************************)

	IF ioMap.In.ModuleOk AND dataInv.Parameters.CommsType = COMMS_POWERLINK THEN
		IF dataInv.Parameters.Type = INV_ABB THEN
			(* Control mode setting with the correct units *)
			ioMap.Out.ControlMode	:= dataInv.Parameters.ControlMode;

			IF dataInv.Parameters.ControlMode = CONTROL_MODE_VECTOR THEN
				ioMap.Out.SpeedUnit		:= 4; // 4 = Control by Speed
				ioMap.Out.AccTimeVector	:= REAL_TO_DINT(dataInv.Parameters.AccelerationTime);
				ioMap.Out.DecTimeVector	:= REAL_TO_DINT(dataInv.Parameters.DecelerationTime);
				ioMap.Out.SetSpeed		:= UINT_TO_INT(dataInv.Parameters.Velocity) * direction;
			ELSIF dataInv.Parameters.ControlMode = CONTROL_MODE_SCALAR THEN
				ioMap.Out.SpeedUnit		:= 5; // 5 = Control by Speed
				ioMap.Out.AccTimeScalar	:= REAL_TO_DINT(dataInv.Parameters.AccelerationTime * RAMP_MAX_HZ_VALUE / (dataInv.Parameters.Velocity * 100.0));
				ioMap.Out.DecTimeScalar	:= REAL_TO_DINT(dataInv.Parameters.DecelerationTime * RAMP_MAX_HZ_VALUE / (dataInv.Parameters.Velocity * 100.0));
				ioMap.Out.SetFrequency	:= UINT_TO_INT(dataInv.Parameters.Velocity * 100) * direction;
			END_IF
			ACC_Ok := TRUE;
			DEC_Ok := TRUE;
		ELSE

			(* Acceleration *)
			dataInv.Parameters.AccelerationTime := LIMIT(ACC_min, dataInv.Parameters.AccelerationTime, ACC_max);	(* Check value *)
			CASE stepTransferACC OF

				0: (* Read parameter *)

					EplSDORead_ACC.pDevice := ADR(PL_device);
					EplSDORead_ACC.node := HW_node;
					EplSDORead_ACC.index := 16#203C;
					EplSDORead_ACC.subindex := 16#02;
					EplSDORead_ACC.pData := ADR(AccTime_actual);
					EplSDORead_ACC.datalen := SIZEOF(AccTime_actual);
					EplSDORead_ACC.enable := TRUE;
					EplSDORead_ACC();
					IF EplSDORead_ACC.status = 0 THEN
						stepTransferACC := 1;
					ELSIF EplSDORead_ACC.status <> ERR_FUB_BUSY THEN
						invalidHwAddress := TRUE;
					END_IF

				1: (* Check change *)
					IF REAL_TO_UINT(dataInv.Parameters.AccelerationTime * 10) = AccTime_actual THEN
						ACC_Ok := TRUE;
					ELSE
						ACC_Ok := FALSE;
						AccTime_set := REAL_TO_UINT(dataInv.Parameters.AccelerationTime * 10);
						stepTransferACC := 2;
					END_IF

				2: (* Write parameter *)

					EplSDOWrite_ACC.pDevice := ADR(PL_device);
					EplSDOWrite_ACC.node := HW_node;
					EplSDOWrite_ACC.index := 16#203C;
					EplSDOWrite_ACC.subindex := 16#02;
					EplSDOWrite_ACC.pData := ADR(AccTime_set);
					EplSDOWrite_ACC.datalen := SIZEOF(AccTime_set);
					EplSDOWrite_ACC.enable := TRUE;
					EplSDOWrite_ACC();
					IF EplSDOWrite_ACC.status = 0 THEN
						stepTransferACC := 0;
					ELSIF EplSDOWrite_ACC.status <> ERR_FUB_BUSY THEN
						invalidHwAddress := TRUE;
					END_IF

			END_CASE

			(* Deceleration *)
			dataInv.Parameters.DecelerationTime := LIMIT(DEC_min, dataInv.Parameters.DecelerationTime, DEC_max);	(* Check value *)
			CASE stepTransferDEC OF

				0: (* Read parameter *)

					EplSDORead_DEC.pDevice := ADR(PL_device);
					EplSDORead_DEC.node := HW_node;
					EplSDORead_DEC.index := 16#203C;
					EplSDORead_DEC.subindex := 16#03;
					EplSDORead_DEC.pData := ADR(DecTime_actual);
					EplSDORead_DEC.datalen := SIZEOF(DecTime_actual);
					EplSDORead_DEC.enable := TRUE;
					EplSDORead_DEC();
					IF EplSDORead_DEC.status = 0 THEN
						stepTransferDEC := 1;
					ELSIF EplSDORead_DEC.status <> ERR_FUB_BUSY THEN
						invalidHwAddress := TRUE;
					END_IF

				1: (* Check change *)
					IF REAL_TO_UINT(dataInv.Parameters.DecelerationTime * 10) = DecTime_actual THEN
						DEC_Ok := TRUE;
					ELSE
						DEC_Ok := FALSE;
						DecTime_set := REAL_TO_UINT(dataInv.Parameters.DecelerationTime * 10);
						stepTransferDEC := 2;
					END_IF

				2: (* Write parameter *)

					EplSDOWrite_DEC.pDevice := ADR(PL_device);
					EplSDOWrite_DEC.node := HW_node;
					EplSDOWrite_DEC.index := 16#203C;
					EplSDOWrite_DEC.subindex := 16#03;
					EplSDOWrite_DEC.pData := ADR(DecTime_set);
					EplSDOWrite_DEC.datalen := SIZEOF(DecTime_set);
					EplSDOWrite_DEC.enable := TRUE;
					EplSDOWrite_DEC();
					IF EplSDOWrite_DEC.status = 0 THEN
						stepTransferDEC := 0;
					ELSIF EplSDOWrite_DEC.status <> ERR_FUB_BUSY THEN
						invalidHwAddress := TRUE;
					END_IF

			END_CASE

		END_IF;

	ELSIF dataInv.Parameters.CommsType = COMMS_CANOPEN THEN
		ACC_Ok := TRUE;
		DEC_Ok := TRUE;
	END_IF

	paramOk := ACC_Ok AND DEC_Ok;
	IF paramOk THEN
		invalidHwAddress := FALSE;
	END_IF

(********************************************************************
	Simulation
*********************************************************************)

	IF dataInv.Parameters.Hardware.CpuFamily = FAMILY_BRAUTOMATIONRUNTIME OR xForceSim THEN
		Simulation;
	END_IF;

(********************************************************************
	Control Handling
*********************************************************************)

	(* Gets the status from the drive *)
	IF ioMap.In.ModuleOk AND (ioMap.In.StatusWord <> 0) AND NOT(connectionErrorNotAck) THEN
		IF ((ioMap.In.StatusWord AND 16#006F) = 16#0000) THEN
			axisStep := STATE_NOT_READY_TO_SWITCH_ON;
		ELSIF ((ioMap.In.StatusWord AND 16#004F) = 16#0040) THEN
			axisStep := STATE_SWITCH_ON_DISABLED;
		ELSIF ((ioMap.In.StatusWord AND 16#006F) = 16#0021) THEN
			axisStep := STATE_READY_TO_SWITCH_ON;
		ELSIF ((ioMap.In.StatusWord AND 16#006F) = 16#0023) THEN
			axisStep := STATE_SWITCHED_ON;
		ELSIF ((ioMap.In.StatusWord AND 16#006F) = 16#0027) THEN
			axisStep := STATE_OPERATION_ENABLED;
		ELSIF ((ioMap.In.StatusWord AND 16#006F) = 16#0007) THEN
			axisStep := STATE_QUICK_STOP_ACTIVE;
		ELSIF ((ioMap.In.StatusWord AND 16#004F) = 16#000F) THEN
			axisStep := STATE_FAULT_REACTION_ACTIVE;
		ELSIF ((ioMap.In.StatusWord AND 16#004F) = 16#0008) THEN
			axisStep := STATE_FAULT;
		ELSE 	(* Connection error or drive malfunction *)
			axisStep := STATE_ERROR;
		END_IF
	ELSE
		IF dataInv.Parameters.CommsType = COMMS_POWERLINK THEN
			ACC_Ok := FALSE;	(* The parameter might have changed *)
			stepTransferACC := 0;	(* Read parameter *)
			DEC_Ok := FALSE;	(* The parameter might have changed *)
			stepTransferDEC := 0;	(* Read parameter *)
			connectionErrorNotAck := TRUE;
		END_IF
		axisStep := STATE_ERROR;

	END_IF

	IF axisStep <> STATE_FAULT THEN
		IF axisStep <> STATE_ERROR THEN
			dataInv.Commands.Reset := FALSE;
		END_IF
		resetCount := 0;
	END_IF

	(* State machine *)
	CASE axisStep OF

(**************************** NOT READY ****************************)
		STATE_NOT_READY_TO_SWITCH_ON:

			IF dataInv.Parameters.Type = INV_ABB THEN
				ioMap.Out.ControlWord := 16#0406;
			ELSE
				ioMap.Out.ControlWord := 16#0000;
			END_IF

(***************************** DISABLED ****************************)
		STATE_SWITCH_ON_DISABLED:
			IF dataInv.Parameters.Type = INV_ABB THEN
				ioMap.Out.ControlWord := 16#0406;
			ELSE
				ioMap.Out.ControlWord := 16#0006;
			END_IF

(****************************** READY ******************************)
		STATE_READY_TO_SWITCH_ON:

			IF (dataInv.Orders.PowerOn) THEN
				IF dataInv.Parameters.Type = INV_ABB THEN
					ioMap.Out.ControlWord := 16#0407;
				ELSE
					ioMap.Out.ControlWord := 16#0007;
				END_IF
			END_IF

(*************************** SWITCHED ON ***************************)
		STATE_SWITCHED_ON:

			IF NOT(dataInv.Orders.PowerOn) THEN
				IF dataInv.Parameters.Type = INV_ABB THEN
					ioMap.Out.ControlWord := 16#0406;
				ELSE
					ioMap.Out.ControlWord := 16#0006;
				END_IF
			ELSIF paramOk THEN
				IF dataInv.Commands.Stop THEN
					direction := 0;
					IF dataInv.Parameters.Type = INV_ABB THEN
						ioMap.Out.ControlWord := 16#0477;
					ELSE
						ioMap.Out.ControlWord := 16#0007;
					END_IF
					dataInv.Commands.MovePositive := FALSE;
					dataInv.Commands.MoveNegative := FALSE;
					dataInv.Commands.Stop := FALSE;
					uiTimesCommandStop := uiTimesCommandStop + 1;
				ELSIF dataInv.Commands.MovePositive THEN
					direction := 1;
					IF dataInv.Parameters.Type = INV_ABB THEN
						ioMap.Out.ControlWord := 16#047F;
					ELSE
						ioMap.Out.ControlWord := 16#000F;
					END_IF
					dataInv.Commands.MovePositive := FALSE;
					uiTimesCommandPositive := uiTimesCommandPositive + 1;
				ELSIF dataInv.Commands.MoveNegative THEN
					direction := -1;
					IF dataInv.Parameters.Type = INV_ABB THEN
						ioMap.Out.ControlWord := 16#047F;
					ELSE
						ioMap.Out.ControlWord := 16#000F;
					END_IF
					dataInv.Commands.MoveNegative := FALSE;
					uiTimesCommandNegative := uiTimesCommandNegative + 1;
				END_IF
			END_IF

(************************ OPERATION_ENABLED ************************)
		STATE_OPERATION_ENABLED:

			IF NOT(dataInv.Orders.PowerOn) THEN
				IF dataInv.Parameters.Type = INV_ABB THEN
					ioMap.Out.ControlWord := 16#0406;
				ELSE
					ioMap.Out.ControlWord := 16#0006;
				END_IF
				dataInv.Commands.MovePositive := FALSE;
				dataInv.Commands.MoveNegative := FALSE;
				dataInv.Commands.Stop := FALSE;
			ELSIF dataInv.Commands.Stop THEN
				direction := 0;
				IF dataInv.Parameters.Type = INV_ABB THEN
					ioMap.Out.ControlWord := 16#0477;
				ELSE
					ioMap.Out.ControlWord := 16#0007; //In CanOpen: ioMap.Out.ControlWord := 16#100F;	(* Stops the axis as configured in FUN->STC->STT (Default: RMP) *)
				END_IF;
				dataInv.Commands.MovePositive := FALSE;
				dataInv.Commands.MoveNegative := FALSE;
				dataInv.Commands.Stop := FALSE;
				uiTimesCommandStop := uiTimesCommandStop + 1;
			ELSIF dataInv.Commands.MovePositive THEN
				direction := 1;
				IF dataInv.Parameters.Type = INV_ABB THEN
					ioMap.Out.ControlWord := 16#047F;
				ELSE
					ioMap.Out.ControlWord := 16#000F;
				END_IF
				dataInv.Commands.MovePositive := FALSE;
				uiTimesCommandPositive := uiTimesCommandPositive + 1;
			ELSIF dataInv.Commands.MoveNegative THEN
				direction := -1;
				IF dataInv.Parameters.Type = INV_ABB THEN
					ioMap.Out.ControlWord := 16#047F;
				ELSE
					ioMap.Out.ControlWord := 16#000F;
				END_IF
				dataInv.Commands.MoveNegative := FALSE;
				uiTimesCommandNegative := uiTimesCommandNegative + 1;
			END_IF

			(* Needed to be compatible with the logical state machine *)
			IF direction = 0 THEN	(* If a stop has been requested *)
				IF ioMap.In.ActualSpeed = 0 THEN	(* If axis is in standstill *)
					ioMap.Out.ControlWord := 16#0007;	(* Returns the inverter to STATE_SWITCHED_ON *)
				END_IF
			END_IF

(************************ QUICK STOP ACTIVE ************************)
		STATE_QUICK_STOP_ACTIVE:

			ioMap.Out.ControlWord := 16#0000;

(************************** FAULT REACTION *************************)
		STATE_FAULT_REACTION_ACTIVE:

			(* Wait until STATE_FAULT *)

(********************** ERROR AND ACKNOWLEDGE **********************)
		STATE_FAULT:

			IF (dataInv.Commands.Reset) THEN
				ioMap.Out.ControlWord := 16#0080;
				resetCount := 1;
				partialCount := 0;
				dataInv.Commands.Reset := FALSE;
			END_IF
			(* Makes a period-increasing Flip-Flop to ensure that the inverter gets a pos. edge *)
			IF resetCount > 0 THEN
				IF partialCount >= resetCount THEN
					ioMap.Out.ControlWord := ioMap.Out.ControlWord XOR 16#0080;
					resetCount := resetCount + 2;
					partialCount := 0;
				ELSE
					partialCount := partialCount + 1;
				END_IF
				IF resetCount >= 24 THEN
					resetCount := 1;
					partialCount := 0;
				END_IF
			END_IF

(************************* CONNECTION ERROR ************************)
		STATE_ERROR:
			IF dataInv.Parameters.Type = INV_ABB THEN
				ioMap.Out.ControlWord := 16#0000;
			END_IF
			IF (dataInv.Commands.Reset) THEN
				connectionErrorNotAck := FALSE;
				dataInv.Commands.Reset := FALSE;
			END_IF

	END_CASE

(********************************************************************
	Speed and Direction Handling
*********************************************************************)

	(* Sets the speed *)
	ioMap.Out.SetSpeed := UINT_TO_INT(dataInv.Parameters.Velocity) * direction;

(*****************************************************************
	Status Handling
******************************************************************)

	(* Reports the drive state *)
	dataInv.Status.ErrorComms			:= NOT ioMap.In.ModuleOk;
	dataInv.Status.StatusDisabled		:= (axisStep = STATE_NOT_READY_TO_SWITCH_ON) OR (axisStep = STATE_SWITCH_ON_DISABLED) OR (axisStep = STATE_READY_TO_SWITCH_ON);
	dataInv.Status.StatusReady			:= (axisStep = STATE_SWITCHED_ON);
	dataInv.Status.StatusOperation		:= (axisStep = STATE_OPERATION_ENABLED) OR (axisStep = STATE_QUICK_STOP_ACTIVE);
	dataInv.Status.StatusErrorStop		:= (axisStep = STATE_FAULT) OR (axisStep = STATE_FAULT_REACTION_ACTIVE) OR (axisStep = STATE_ERROR);
	dataInv.Status.ReadyForOrders		:=  dataInv.Orders.PowerOn AND ((axisStep = STATE_SWITCHED_ON AND paramOk) OR (axisStep = STATE_OPERATION_ENABLED)); //Adding dataInv.Orders.PowerOn and paramOk here because is when we are really ready to receive orders

	(* Reports errors *)
	IF dataInv.Parameters.Type = INV_ABB THEN
		ErrMessage_FUB.CurrentErrID		:= ioMap.In.ErrorID;

		IF axisStep = STATE_FAULT THEN
			dataInv.Status.ErrorID 		:= INT_TO_UINT(ioMap.In.ErrorID);
			dataInv.Status.ErrorText 	:= ErrMessage_FUB.CurrentErrMessage;
			ErrMessage_FUB.NewID		:= TRUE;
		ELSIF axisStep = STATE_ERROR THEN
			dataInv.Status.ErrorID 		:= 7510;
			dataInv.Status.ErrorText 	:= 'Communication error';
			ioMap.Out.Reset				:= dataInv.Commands.Reset;
		ELSE
			dataInv.Status.ErrorID	 	:= 0;
			dataInv.Status.ErrorText 	:= '';
			ioMap.Out.Reset				:= 0;
			dataInv.Commands.Reset		:= 0;
		END_IF
		(* Error message *)
		ErrMessage_FUB();

	ELSE
		IF axisStep = STATE_FAULT THEN
			dataInv.Status.ErrorID := INT_TO_UINT(ioMap.In.ErrorID);
			dataInv.Status.ErrorText := ERROR_TEXT[LIMIT(0, dataInv.Status.ErrorID, 109)];
		ELSIF axisStep = STATE_ERROR THEN
			dataInv.Status.ErrorID := 50034;
			dataInv.Status.ErrorText := 'SLF1/COF';
		ELSIF invalidHwAddress THEN
			dataInv.Status.ErrorID := 51000;
			dataInv.Status.ErrorText := 'Invalid HW Address';
		ELSE
			dataInv.Status.ErrorID := 0;
			dataInv.Status.ErrorText := '';
		END_IF
	END_IF
	(* Reports the actual speed *)
	dataInv.Status.ActVelocity := ioMap.In.ActualSpeed;
	dataInv.Status.xAtSpeed := ABS(ABS(dataInv.Status.ActVelocity)-dataInv.Parameters.Velocity)<(dataInv.Parameters.Velocity/100);

	(* Reports the actual current *)
	IF dataInv.Parameters.Type = INV_ABB THEN
		dataInv.Status.ActCurrent := INT_TO_REAL(ioMap.In.ActualCurrentABB)/ 1000;
	ELSE
		dataInv.Status.ActCurrent := UINT_TO_REAL(ioMap.In.ActualCurrent)/ 10;
	END_IF
	(* Reports the actual Torque *)
	dataInv.Status.ActTorque := INT_TO_REAL(ioMap.In.ActualTorque)/10;

	//In CanOpen, acceleration and deceleration by PDO
	IF dataInv.Parameters.CommsType = COMMS_CANOPEN THEN

		(* Acceleration *)
		dataInv.Parameters.AccelerationTime := LIMIT(ACC_min, dataInv.Parameters.AccelerationTime, ACC_max); (* Check value *)
		ioMap.Out.Acceleration := REAL_TO_UINT(dataInv.Parameters.AccelerationTime * 10);

		(* Deceleration *)
		dataInv.Parameters.DecelerationTime := LIMIT(DEC_min, dataInv.Parameters.DecelerationTime, DEC_max); (* Check value *)
		ioMap.Out.Deceleration := REAL_TO_UINT(dataInv.Parameters.DecelerationTime * 10);

	END_IF

	IF dataInv.Parameters.CommsType = COMMS_POWERLINK THEN

		(* Reports the state of the digital inputs*)
		dataInv.DigitalInput[0] := ioMap.In.DigitalInput[0];
		dataInv.DigitalInput[1] := ioMap.In.DigitalInput[1];
		dataInv.DigitalInput[2] := ioMap.In.DigitalInput[2];
		dataInv.DigitalInput[3] := ioMap.In.DigitalInput[3];
		dataInv.DigitalInput[4] := ioMap.In.DigitalInput[4];
		dataInv.DigitalInput[5] := ioMap.In.DigitalInput[5];
		dataInv.DigitalInput[6] := ioMap.In.DigitalInput[6];
		dataInv.DigitalInput[7] := ioMap.In.DigitalInput[7];

		(* Reports the state of the digital outputs*)
		ioMap.Out.DigitalOutput[0] := dataInv.DigitalOutput[0];
		ioMap.Out.DigitalOutput[1] := dataInv.DigitalOutput[1];
		ioMap.Out.DigitalOutput[2] := dataInv.DigitalOutput[2];

		(* Reports the state of the digital outputs*)
		ioMap.Out.AnalogOutput := dataInv.AnalogOutput;

	ELSIF dataInv.Parameters.CommsType = COMMS_CANOPEN THEN

		(* Reports the state of the digital inputs*)
		dataInv.DigitalInput[0] := ioMap.In.DigitalInputs.0;
		dataInv.DigitalInput[1] := ioMap.In.DigitalInputs.1;
		dataInv.DigitalInput[2] := ioMap.In.DigitalInputs.2;
		dataInv.DigitalInput[3] := ioMap.In.DigitalInputs.3;
		dataInv.DigitalInput[4] := ioMap.In.DigitalInputs.4;
		dataInv.DigitalInput[5] := ioMap.In.DigitalInputs.5;

		(* Reports the state of the digital outputs*)
		ioMap.Out.DigitalOutputs.0 := dataInv.DigitalOutput[0]; //RELAY
		ioMap.Out.DigitalOutputs.1 := dataInv.DigitalOutput[1]; //RELAY
		ioMap.Out.DigitalOutputs.8 := dataInv.DigitalOutput[2];

		(* Reports the state of the digital outputs*)
		ioMap.Out.AnalogOutputSigned := dataInv.AnalogOutput;

	END_IF

	(* Reports the state of the digital inputs*)
	dataInv.AnalogInput := ioMap.In.AnalogInput;

//	//Get CANOpen state
//	CanGetState.enable := TRUE;
//	CanGetState.node := dataInv.Parameters.Hardware.Node;
//	CanGetState.pDevice := ADR('SS1.IF1');
//	CanGetState();

END_ACTION
```

#### InverterCtrl.var - Local variables
```iecst
(********************************************************************
 * COPYRIGHT -- Bernecker + Rainer
 ********************************************************************
 * Program: I66Ctrl
 * File: I66Ctrl.var
 * Author: tresensa
 * Created: May 09, 2014
 ********************************************************************
 * Local variables of program I66Ctrl
 ********************************************************************)
(* *******************************************************************
 * data Reference
 ********************************************************************)
VAR
	dataInv : REFERENCE TO AxisP66_typ; (*I/O Mapping for the ACOPOSinverter*)
END_VAR
(* *******************************************************************
 * IO Mapping
 ********************************************************************)
VAR
	ioMap : REFERENCE TO AxisP66_Signals_typ; (*I/O Mapping for the ACOPOSinverter*)
END_VAR
(* *******************************************************************
 * State Machine
 ********************************************************************)
VAR
	axisStep : UINT;
END_VAR
VAR CONSTANT
	STATE_NOT_READY_TO_SWITCH_ON : USINT := 1;
	STATE_SWITCH_ON_DISABLED : USINT := 2;
	STATE_READY_TO_SWITCH_ON : USINT := 3;
	STATE_SWITCHED_ON : USINT := 4;
	STATE_OPERATION_ENABLED : USINT := 5;
	STATE_QUICK_STOP_ACTIVE : USINT := 6;
	STATE_FAULT_REACTION_ACTIVE : USINT := 7;
	STATE_FAULT : USINT := 8;
	STATE_ERROR : USINT := 100;
END_VAR
(* *******************************************************************
 * Error Texts
 ********************************************************************)
VAR
	ERROR_TEXT : ARRAY[0..109] OF STRING[19]; (*Table of error descriptions*)
	Error : ARRAY[0..199] OF Errors_type;
END_VAR
(* *******************************************************************
 * Temp
 ********************************************************************)
VAR
	resetCount : UINT;
	partialCount : UINT;
	direction : SINT;
END_VAR
(* *******************************************************************
 * Control Modes
 ********************************************************************)
VAR CONSTANT
	CONTROL_MODE_VECTOR : UINT := 0;
	CONTROL_MODE_SCALAR : UINT := 1;
	RAMP_MAX_SPEED_VALUE : DINT := 2000000;
END_VAR
VAR
	ErrMessage_FUB : ErrMessage;
END_VAR
VAR CONSTANT
	RAMP_MAX_HZ_VALUE : UDINT := 20000;
END_VAR
(* *******************************************************************
 * Parameter Transfer
 ********************************************************************)
VAR
	PL_device : STRING[39]; (*Physical address of the Powerlink IF*)
	HW_node : USINT; (*Inverter's Powerlink node*)
END_VAR
VAR CONSTANT
	ACC_min : REAL := 0.1; (*(From datasheet)*)
	ACC_max : REAL := 999.9; (*(From datasheet)*)
	DEC_min : REAL := 0.1; (*(From datasheet)*)
	DEC_max : REAL := 999.9; (*(From datasheet)*)
END_VAR
VAR
	stepTransferACC : USINT := 0;
	stepTransferDEC : USINT := 0;
	AccTime_actual : UINT;
	DecTime_actual : UINT;
	AccTime_set : UINT;
	DecTime_set : UINT;
	ACC_Ok : BOOL;
	DEC_Ok : BOOL;
	paramOk : BOOL;
	invalidHwAddress : BOOL;
	EplSDORead_ACC : EplSDORead;
	EplSDOWrite_ACC : EplSDOWrite;
	EplSDORead_DEC : EplSDORead;
	EplSDOWrite_DEC : EplSDOWrite;
	connectionErrorNotAck : BOOL;
END_VAR
(* *******************************************************************
 * Parameter Simulation
 ********************************************************************)
VAR
	StepSim : USINT := 1; (*State machine for simulation*)
	SimNominalSpeed : UINT := 3000; (*Motor nominal speed [rpm]*)
	SimCycleTime : REAL := 0.002; (*Cycle time of the task [s]*)
	SimVelocity : REAL;
	SimInitialVelocity : REAL;
	SimAcceleration : REAL;
	SimDecceleration : REAL;
	RTInfo_0 : RTInfo;
	xForceSim : BOOL; (*Local variable to enable simulation with REAL PLC*)
	uiTimesCommandStop : UINT;
	uiTimesCommandPositive : UINT;
	uiTimesCommandNegative : UINT;
	CanGetState : CANopenGetState;
	tonNotComms : TON;
	tonCommsErrorResetting : TON;
	CanResetState : CanOpenResetCommsState_enum;
	CanResetState_copy : CanOpenResetCommsState_enum;
	CANopenReset : CANopenNMT;
	iReasonNotComms : UINT;
	xChangedResetCommsState : BOOL;
	lastResetingState : UINT;
	lastFbResetStatus : UINT;
	lastCanOpenResetError : UINT;
	iTimesTryToReset : UINT;
END_VAR
```

#### ErrorTableACS380.st
```iecst
(*************************************************************************
 * COPYRIGHT -- Bernecker + Rainer
 *************************************************************************
 * Program: ACS380Ctrl
 * File: ErrorTable.st
 * Author: canyisc
 * Created: April 24, 2019
 *************************************************************************
 * ERRORS and WARNINGS OF program ABB ACS380
 *************************************************************************
 *************************************************************************
 * Version | Date			| Author 	| Description
 * ----------------------------------------------------------------------
 * V1.00.0 | 17-April-2019 	| canyisc	| Adapted TO ABB ACS380 inverter
 ************************************************************************)

(*Writes the error table*)
ACTION ErrorTableACS380:

	// ----------------------------------------------------------------------------------------
	// 								FAULT MESSAGES
	// ----------------------------------------------------------------------------------------

	Error[0].ErrorID	:= 16#1080;
	Error[0].ErrorText	:= 'Err 1080: Backup/Restore timeout';

	Error[1].ErrorID	:= 16#1081;
	Error[1].ErrorText	:= 'Err 1081: Rating ID fault';

	Error[2].ErrorID	:= 16#2281;
	Error[2].ErrorText	:= 'Err 2281: Calibration';

	Error[3].ErrorID	:= 16#2310;
	Error[3].ErrorText	:= 'Err 2310: Overcurrent';

	Error[4].ErrorID	:= 16#2330;
	Error[4].ErrorText	:= 'Err 2330: Earth leakage';

	Error[5].ErrorID	:= 16#2340;
	Error[5].ErrorText	:= 'Err 2340: Short circuit';

	Error[6].ErrorID	:= 16#2381;
	Error[6].ErrorText	:= 'Err 2381: IGBT overload';

	Error[7].ErrorID	:= 16#3130;
	Error[7].ErrorText	:= 'Err 3130: Input phase loss';

	Error[8].ErrorID	:= 16#3181;
	Error[8].ErrorText	:= 'Err 3181: Cross connection';

	Error[9].ErrorID	:= 16#3210;
	Error[9].ErrorText	:= 'Err 3210: DC link overvoltage';

	Error[10].ErrorID	:= 16#3220;
	Error[10].ErrorText	:= 'Err 3220: DC link undervoltage';

	Error[11].ErrorID	:= 16#3385;
	Error[11].ErrorText	:= 'Err 3385: Autophasing';

	Error[12].ErrorID	:= 16#3381;
	Error[12].ErrorText	:= 'Err 3381: Output phase loss';

	Error[13].ErrorID	:= 16#4110;
	Error[13].ErrorText	:= 'Err 4110: Control board temperature';

	Error[14].ErrorID	:= 16#4210;
	Error[14].ErrorText	:= 'Err 4210: IGBT overtemperature';

	Error[15].ErrorID	:= 16#4290;
	Error[15].ErrorText	:= 'Err 4290: Cooling';

	Error[16].ErrorID	:= 16#42F1;
	Error[16].ErrorText	:= 'Err 42F1: IGBT temperature';

	Error[17].ErrorID	:= 16#4310;
	Error[17].ErrorText	:= 'Err 4310: Excess temperature';

	Error[18].ErrorID	:= 16#4380;
	Error[18].ErrorText	:= 'Err : Excess temperature difference';

	Error[19].ErrorID	:= 16#4981;
	Error[19].ErrorText	:= 'Err 4380: External temperature 1';

	Error[20].ErrorID	:= 16#4982;
	Error[20].ErrorText	:= 'Err 4982: External temperature 2';

	Error[21].ErrorID	:= 16#5090;
	Error[21].ErrorText	:= 'Err 5090: STO hardware failure';

	Error[22].ErrorID	:= 16#5091;
	Error[22].ErrorText	:= 'Err 5091: Safe torque off';

	Error[23].ErrorID	:= 16#5092;
	Error[23].ErrorText	:= 'Err 5092: PU logic error';

	Error[24].ErrorID	:= 16#5093;
	Error[24].ErrorText	:= 'Err 5093: Rating ID mismatch';

	Error[25].ErrorID	:= 16#5094;
	Error[25].ErrorText	:= 'Err 5094: Measurement circuit temperature';

	Error[26].ErrorID	:= 16#5098;
	Error[26].ErrorText	:= 'Err 5098: I/O communication loss';

	Error[27].ErrorID	:= 16#50A0;
	Error[27].ErrorText	:= 'Err 50A0: Fan';

	Error[28].ErrorID	:= 16#5681;
	Error[28].ErrorText	:= 'Err 5681: PU communication';

	Error[29].ErrorID	:= 16#5682;
	Error[29].ErrorText	:= 'Err 5682: Power unit lost';

	Error[30].ErrorID	:= 16#5690;
	Error[30].ErrorText	:= 'Err 5690: PU communication internal';

	Error[31].ErrorID	:= 16#5691;
	Error[31].ErrorText	:= 'Err 5691: Measurement circuit ADC';

	Error[32].ErrorID	:= 16#5692;
	Error[32].ErrorText	:= 'Err 5692: PU board powerfail';

	Error[33].ErrorID	:= 16#5693;
	Error[33].ErrorText	:= 'Err 5693: Measurement circuit DFF';

	Error[34].ErrorID	:= 16#5696;
	Error[34].ErrorText	:= 'Err 5696: PU state feedback';

	Error[35].ErrorID	:= 16#5697;
	Error[35].ErrorText	:= 'Err 5697: Charging feedback';

	Error[36].ErrorID	:= 16#6181;
	Error[36].ErrorText	:= 'Err 6181: FPGA version incompatible';

	Error[37].ErrorID	:= 16#6200;
	Error[37].ErrorText	:= 'Err 6200: Checksum mismatch';

	Error[38].ErrorID	:= 16#6306;
	Error[38].ErrorText	:= 'Err 6306: FBA A mapping file';

	Error[39].ErrorID	:= 16#6481;
	Error[39].ErrorText	:= 'Err 6481: Task overload';

	Error[40].ErrorID	:= 16#6487;
	Error[40].ErrorText	:= 'Err 6487: Stack overflow';

	Error[41].ErrorID	:= 16#64A1;
	Error[41].ErrorText	:= 'Err 64A1: Internal file load';

	Error[42].ErrorID	:= 16#64A6;
	Error[42].ErrorText	:= 'Err 64A6: Adaptive program file incompatible OR corrupted';

	Error[43].ErrorID	:= 16#64B2;
	Error[43].ErrorText	:= 'Err 64B2: User set fault';

	Error[44].ErrorID	:= 16#64E1;
	Error[44].ErrorText	:= 'Err 64E1: Kernel overload';

	Error[45].ErrorID	:= 16#6581;
	Error[45].ErrorText	:= 'Err 6581: Parameter system';

	Error[46].ErrorID	:= 16#65A1;
	Error[46].ErrorText	:= 'Err 65A1: FBA A parameter conflict';

	Error[47].ErrorID	:= 16#6681;
	Error[47].ErrorText	:= 'Err 6681: EFB comm loss';

	Error[48].ErrorID	:= 16#6682;
	Error[48].ErrorText	:= 'Err 6682: EFB config file';

	Error[49].ErrorID	:= 16#6683;
	Error[49].ErrorText	:= 'Err 6683: EFB invalid parameterization';

	Error[50].ErrorID	:= 16#6684;
	Error[50].ErrorText	:= 'Err 6684: EFB load fault';

	Error[51].ErrorID	:= 16#6685;
	Error[51].ErrorText	:= 'Err 6685: EFB fault 2';

	Error[52].ErrorID	:= 16#6686;
	Error[52].ErrorText	:= 'Err 6686: EFB fault 3';

	Error[53].ErrorID	:= 16#6882;
	Error[53].ErrorText	:= 'Err 6882: Text 32-bit table overflow';

	Error[54].ErrorID	:= 16#6885;
	Error[54].ErrorText	:= 'Err 6885: Text file overflow';

	Error[55].ErrorID	:= 16#7081;
	Error[55].ErrorText	:= 'Err 7081: Control panel loss';

	Error[56].ErrorID	:= 16#7082;
	Error[56].ErrorText	:= 'Err 7082: I/O module comm loss';

	Error[57].ErrorID	:= 16#7086;
	Error[57].ErrorText	:= 'Err 7086: I/O module AI Over voltage';

	Error[58].ErrorID	:= 16#71A2;
	Error[58].ErrorText	:= 'Err 71A2: Mechanical brake closing failed';

	Error[59].ErrorID	:= 16#71A3;
	Error[59].ErrorText	:= 'Err 71A3: Mechanical brake opening failed';

	Error[60].ErrorID	:= 16#71A5;
	Error[60].ErrorText	:= 'Err 71A5: Mechanical brake opening NOT allowed';

	Error[61].ErrorID	:= 16#7121;
	Error[61].ErrorText	:= 'Err 7121: Motor stall';

	Error[62].ErrorID	:= 16#7181;
	Error[62].ErrorText	:= 'Err 7181: Brake resistor';

	Error[63].ErrorID	:= 16#7183;
	Error[63].ErrorText	:= 'Err 7183: BR excess temperature';

	Error[64].ErrorID	:= 16#7184;
	Error[64].ErrorText	:= 'Err 7184: Brake resistor wiring';

	Error[65].ErrorID	:= 16#7191;
	Error[65].ErrorText	:= 'Err 7191: BC short circuit';

	Error[66].ErrorID	:= 16#7192;
	Error[66].ErrorText	:= 'Err 7192: BC IGBT excess temperature';

	Error[67].ErrorID	:= 16#7301;
	Error[67].ErrorText	:= 'Err 7301: Motor speed feedback';

	Error[68].ErrorID	:= 16#7310;
	Error[68].ErrorText	:= 'Err 7310: Overspeed';

	Error[69].ErrorID	:= 16#7381;
	Error[69].ErrorText	:= 'Err 7381: Encoder';

	Error[70].ErrorID	:= 16#73F0;
	Error[70].ErrorText	:= 'Err 73F0: Overfrequency';

	Error[71].ErrorID	:= 16#73B0;
	Error[71].ErrorText	:= 'Err 73B0: Emergency ramp failed';

	Error[72].ErrorID	:= 16#7510;
	Error[72].ErrorText	:= 'Err 7510: FBA A communication';

	Error[73].ErrorID	:= 16#8001;
	Error[73].ErrorText	:= 'Err 8001: ULC underload fault';

	Error[74].ErrorID	:= 16#8002;
	Error[74].ErrorText	:= 'Err 8002: ULC overload fault';

	Error[75].ErrorID	:= 16#80A0;
	Error[75].ErrorText	:= 'Err 80A0: AI supervision';

	Error[76].ErrorID	:= 16#80B0;
	Error[76].ErrorText	:= 'Err 80B0: Signal supervision';

	Error[77].ErrorID	:= 16#80B1;
	Error[77].ErrorText	:= 'Err 80B1: Signal supervision';

	Error[78].ErrorID	:= 16#80B2;
	Error[78].ErrorText	:= 'Err 80B2: Signal supervision';

	Error[79].ErrorID	:= 16#80B3;
	Error[79].ErrorText	:= 'Err 80B3: Signal supervision';

	Error[80].ErrorID	:= 16#80B4;
	Error[80].ErrorText	:= 'Err 80B4: Signal supervision';

	Error[81].ErrorID	:= 16#80B5;
	Error[81].ErrorText	:= 'Err 80B5: Signal supervision';

	Error[82].ErrorID	:= 16#9081;
	Error[82].ErrorText	:= 'Err 9081: External fault 1';

	Error[83].ErrorID	:= 16#9082;
	Error[83].ErrorText	:= 'Err 9082: External fault 2';

	Error[84].ErrorID	:= 16#9083;
	Error[84].ErrorText	:= 'Err 9083: External fault 3';

	Error[85].ErrorID	:= 16#9084;
	Error[85].ErrorText	:= 'Err 9084: External fault 4';

	Error[86].ErrorID	:= 16#9085;
	Error[86].ErrorText	:= 'Err 9085: External fault 5';

	Error[87].ErrorID	:= 16#FA81;
	Error[87].ErrorText	:= 'Err FA81: Safe torque off 1';

	Error[88].ErrorID	:= 16#FA82;
	Error[88].ErrorText	:= 'Err FA82: Safe torque off 2';

	Error[89].ErrorID	:= 16#FF61;
	Error[89].ErrorText	:= 'Err FF61: ID run';

	Error[90].ErrorID	:= 16#FF81;
	Error[90].ErrorText	:= 'Err FF81: FB A force trip';

	Error[91].ErrorID	:= 16#FF8E;
	Error[91].ErrorText	:= 'Err FF8E: EFB force trip';

	Error[92].ErrorID	:= 16#D100;
	Error[92].ErrorText	:= 'Err D100: Torque prove';

	Error[93].ErrorID	:= 16#D101;
	Error[93].ErrorText	:= 'Err D101: Brake slip';

	Error[94].ErrorID	:= 16#D102;
	Error[94].ErrorText	:= 'Err D102: Brake safe closure';

	Error[95].ErrorID	:= 16#D105;
	Error[95].ErrorText	:= 'Err D105: Speed match';

	Error[96].ErrorID	:= 16#D108;
	Error[96].ErrorText	:= 'Err D108: Stop limits I/O error';

	Error[97].ErrorID	:= 16#D10A;
	Error[97].ErrorText	:= 'Err D10A: Brake not selected';

	// ----------------------------------------------------------------------------------------
	// 								WARNING MESSAGES
	// ----------------------------------------------------------------------------------------

	Error[100].ErrorID		:= 16#64FF;
	Error[100].ErrorText	:= 'Warn 64FF: Fault reset';

	Error[101].ErrorID		:= 16#A2A1;
	Error[101].ErrorText	:= 'Warn A2A1: Current calibration';

	Error[102].ErrorID		:= 16#A2B1;
	Error[102].ErrorText	:= 'Warn A2B1: Overcurrent';

	Error[103].ErrorID		:= 16#A2B3;
	Error[103].ErrorText	:= 'Warn A2B3: Earth leakage';

	Error[104].ErrorID		:= 16#A2B4;
	Error[104].ErrorText	:= 'Warn A2B4: Short circuit';

	Error[105].ErrorID		:= 16#A2B2;
	Error[105].ErrorText	:= 'Warn A2B2: IGBT overload';

	Error[106].ErrorID		:= 16#A3A1;
	Error[106].ErrorText	:= 'Warn A3A1: DC link overvoltage';

	Error[107].ErrorID		:= 16#A3A2;
	Error[107].ErrorText	:= 'Warn A3A2: DC link undervoltage';

	Error[108].ErrorID		:= 16#A3AA;
	Error[108].ErrorText	:= 'Warn A3AA: DC not charged';

	Error[109].ErrorID		:= 16#A490;
	Error[109].ErrorText	:= 'Warn A490: Incorrect temperature sensor setup';

	Error[110].ErrorID		:= 16#A491;
	Error[110].ErrorText	:= 'Warn A491: External temperature 1';

	Error[111].ErrorID		:= 16#A492;
	Error[111].ErrorText	:= 'Warn A492: External temperature 2';

	Error[112].ErrorID		:= 16#A4A1;
	Error[112].ErrorText	:= 'Warn A4A1: IGBT overtemperature';

	Error[113].ErrorID		:= 16#A4A1;
	Error[113].ErrorText	:= 'Warn A4A1: Cooling';

	Error[114].ErrorID		:= 16#A4B0;
	Error[114].ErrorText	:= 'Warn A4B0: Excess temperature';

	Error[115].ErrorID		:= 16#A4B1;
	Error[115].ErrorText	:= 'Warn A4B1: Excess temperature difference';

	Error[116].ErrorID		:= 16#A4F6;
	Error[116].ErrorText	:= 'Warn A4F6: IGBT temperature';

	Error[117].ErrorID		:= 16#A580;
	Error[117].ErrorText	:= 'Warn A580: PU communication';

	Error[118].ErrorID		:= 16#A591;
	Error[118].ErrorText	:= 'Warn A591: Drive HW initialization';

	Error[119].ErrorID		:= 16#A5A0;
	Error[119].ErrorText	:= 'Warn A5A0: Safe torque off';

	Error[120].ErrorID		:= 16#A5EA;
	Error[120].ErrorText	:= 'Warn A5EA: Measurement circuit temperature';

	Error[121].ErrorID		:= 16#A5EB;
	Error[121].ErrorText	:= 'Warn A5EB: PU board powerfail';

	Error[122].ErrorID		:= 16#A5EC;
	Error[122].ErrorText	:= 'Warn A5EC: PU communication internal';

	Error[123].ErrorID		:= 16#A5ED;
	Error[123].ErrorText	:= 'Warn A5ED: Measurement circuit ADC';

	Error[124].ErrorID		:= 16#A5EE;
	Error[124].ErrorText	:= 'Warn A5EE: Measurement circuit DFF';

	Error[125].ErrorID		:= 16#A5EF;
	Error[125].ErrorText	:= 'Warn A5EF: PU state feedback';

	Error[126].ErrorID		:= 16#A5F0;
	Error[126].ErrorText	:= 'Warn A5F0: Charging feedback';

	Error[127].ErrorID		:= 16#A686;
	Error[127].ErrorText	:= 'Warn A686: Checksum mismatch';

	Error[128].ErrorID		:= 16#A687;
	Error[128].ErrorText	:= 'Warn A687: Checksum configuration';

	Error[129].ErrorID		:= 16#A6A4;
	Error[129].ErrorText	:= 'Warn A6A4: Motor nominal value';

	Error[130].ErrorID		:= 16#A6A5;
	Error[130].ErrorText	:= 'Warn A6A5: No motor data';

	Error[131].ErrorID		:= 16#A6A6;
	Error[131].ErrorText	:= 'Warn A6A6: Voltage category unselected';

	Error[132].ErrorID		:= 16#A6B0;
	Error[132].ErrorText	:= 'Warn A6B0: User lock is open';

	Error[133].ErrorID		:= 16#A6D1;
	Error[133].ErrorText	:= 'Warn A6D1: FBA A parameter conflict';

	Error[134].ErrorID		:= 16#A6E5;
	Error[134].ErrorText	:= 'Warn A6E5: AI parametrization';

	Error[135].ErrorID		:= 16#A6E6;
	Error[135].ErrorText	:= 'Warn A6E6: ULC configuration';

	Error[136].ErrorID		:= 16#A7A1;
	Error[136].ErrorText	:= 'Warn A7A1: Mechanical brake closing failed';

	Error[137].ErrorID		:= 16#A7A5;
	Error[137].ErrorText	:= 'Warn A7A5: Mechanical brake opening NOT allowed';

	Error[138].ErrorID		:= 16#A7B0;
	Error[138].ErrorText	:= 'Warn A7B0: Motor speed feedback';

	Error[139].ErrorID		:= 16#A780;
	Error[139].ErrorText	:= 'Warn A780: Motor stall';

	Error[140].ErrorID		:= 16#A791;
	Error[140].ErrorText	:= 'Warn A791: Brake resistor';

	Error[141].ErrorID		:= 16#A793;
	Error[141].ErrorText	:= 'Warn A793: BR excess temperature';

	Error[142].ErrorID		:= 16#A794;
	Error[142].ErrorText	:= 'Warn A794: BR data';

	Error[143].ErrorID		:= 16#A79C;
	Error[143].ErrorText	:= 'Warn A79C: BC IGBT excess temperature';

	Error[144].ErrorID		:= 16#A7AB;
	Error[144].ErrorText	:= 'Warn A7AB: Extension I/O configuration failure';

	Error[145].ErrorID		:= 16#A7C1;
	Error[145].ErrorText	:= 'Warn A7C1: FBA A communication';

	Error[146].ErrorID		:= 16#A7CE;
	Error[146].ErrorText	:= 'Warn A7CE: EFB comm loss';

	Error[147].ErrorID		:= 16#A7E1;
	Error[147].ErrorText	:= 'Warn A7E1: Encoder';

	Error[148].ErrorID		:= 16#A7EE;
	Error[148].ErrorText	:= 'Warn A7EE: Panel loss';

	Error[149].ErrorID		:= 16#A71C;
	Error[149].ErrorText	:= 'Warn A71C: I/O Module internal error';

	Error[150].ErrorID		:= 16#A8A0;
	Error[150].ErrorText	:= 'Warn A8A0: AI supervision';

	Error[151].ErrorID		:= 16#A8A1;
	Error[151].ErrorText	:= 'Warn A8A1: RO life warning';

	Error[152].ErrorID		:= 16#A8A2;
	Error[152].ErrorText	:= 'Warn A8A2: RO toggle warning';

	Error[153].ErrorID		:= 16#A8B0;
	Error[153].ErrorText	:= 'Warn A8B0: Signal supervision';

	Error[154].ErrorID		:= 16#A8B1;
	Error[154].ErrorText	:= 'Warn A8B1: Signal supervision';

	Error[155].ErrorID		:= 16#A8B2;
	Error[155].ErrorText	:= 'Warn A8B2: Signal supervision';

	Error[156].ErrorID		:= 16#A8B3;
	Error[156].ErrorText	:= 'Warn A8B3: Signal supervision';

	Error[157].ErrorID		:= 16#A8B4;
	Error[157].ErrorText	:= 'Warn A8B4: Signal supervision';

	Error[158].ErrorID		:= 16#A8B5;
	Error[158].ErrorText	:= 'Warn A8B5: Signal supervision';

	Error[159].ErrorID		:= 16#A8C0;
	Error[159].ErrorText	:= 'Warn A8C0: ULC invalid speed table';

	Error[160].ErrorID		:= 16#A8C1;
	Error[160].ErrorText	:= 'Warn A8C1: ULC overload warning';

	Error[161].ErrorID		:= 16#A8C4;
	Error[161].ErrorText	:= 'Warn A8C4: ULC underload warning';

	Error[162].ErrorID		:= 16#A8C5;
	Error[162].ErrorText	:= 'Warn A8C5: ULC invalid underload table';

	Error[163].ErrorID		:= 16#A8C6;
	Error[163].ErrorText	:= 'Warn A8C6: ULC invalid overload table';

	Error[164].ErrorID		:= 16#A8C8;
	Error[164].ErrorText	:= 'Warn A8C8: ULC invalid frequency table';

	Error[165].ErrorID		:= 16#A981;
	Error[165].ErrorText	:= 'Warn A981: External warning 1';

	Error[166].ErrorID		:= 16#A982;
	Error[166].ErrorText	:= 'Warn A982: External warning 2';

	Error[167].ErrorID		:= 16#A983;
	Error[167].ErrorText	:= 'Warn A983: External warning 3';

	Error[168].ErrorID		:= 16#A984;
	Error[168].ErrorText	:= 'Warn A984: External warning 4';

	Error[169].ErrorID		:= 16#A985;
	Error[169].ErrorText	:= 'Warn A985: External warning 5';

	Error[170].ErrorID		:= 16#AF88;
	Error[170].ErrorText	:= 'Warn AF88: Season configuration warning';

	Error[171].ErrorID		:= 16#AF8C;
	Error[171].ErrorText	:= 'Warn AF8C: Process PID sleep mode';

	Error[172].ErrorID		:= 16#AFAA;
	Error[172].ErrorText	:= 'Warn AFAA: Autoreset';

	Error[173].ErrorID		:= 16#AFE1;
	Error[173].ErrorText	:= 'Warn AFE1: Emergency stop (off2)';

	Error[174].ErrorID		:= 16#AFE2;
	Error[174].ErrorText	:= 'Warn AFE2: Emergency stop (off1 OR off3)';

	Error[175].ErrorID		:= 16#AFEA;
	Error[175].ErrorText	:= 'Warn AFEA: Enable start signal missing';

	Error[176].ErrorID		:= 16#AFE9;
	Error[176].ErrorText	:= 'Warn AFE9: Start delay';

	Error[177].ErrorID		:= 16#AFEB;
	Error[177].ErrorText	:= 'Warn AFEB: Run enable missing';

	Error[178].ErrorID		:= 16#AFEC;
	Error[178].ErrorText	:= 'Warn AFEC: External power signal missing';

	Error[179].ErrorID		:= 16#AFED;
	Error[179].ErrorText	:= 'Warn AFED: Enable to rotate';

	Error[180].ErrorID		:= 16#AFF6;
	Error[180].ErrorText	:= 'Warn AFF6: Identification run';

	Error[181].ErrorID		:= 16#AFF7;
	Error[181].ErrorText	:= 'Warn AFF7: Autophasing';

	Error[182].ErrorID		:= 16#B5A0;
	Error[182].ErrorText	:= 'Warn B5A0: STO event';

	Error[183].ErrorID		:= 16#B686;
	Error[183].ErrorText	:= 'Warn B686: Checksum mismatch';

	Error[184].ErrorID		:= 16#D200;
	Error[184].ErrorText	:= 'Warn D200: Brake slip at standstill2';

	Error[185].ErrorID		:= 16#D201;
	Error[185].ErrorText	:= 'Warn D201: Forward slow down LIMIT';

	Error[186].ErrorID		:= 16#D202;
	Error[186].ErrorText	:= 'Warn D202: Reverse slow down LIMIT';

	Error[187].ErrorID		:= 16#D205;
	Error[187].ErrorText	:= 'Warn D205: Forward stop limit';

	Error[188].ErrorID		:= 16#D206;
	Error[188].ErrorText	:= 'Warn D206: Reverse stop limit';

	Error[189].ErrorID		:= 16#D208;
	Error[189].ErrorText	:= 'Warn D208: Joystick reference check';

	Error[190].ErrorID		:= 16#D209;
	Error[190].ErrorText	:= 'Warn D209: Joystick zero position';

	Error[191].ErrorID		:= 16#D20A;
	Error[191].ErrorText	:= 'Warn D20A: Fast stop';

	Error[192].ErrorID		:= 16#D20B;
	Error[192].ErrorText	:= 'Warn D20B: Power on acknowledge';

	// ----------------------------------------------------------------------------------------
	// 								NO ERROR MESSAGE
	// ----------------------------------------------------------------------------------------

	Error[199].ErrorID		:= 16#0000;
	Error[199].ErrorText	:= '';

END_ACTION
```

### Program Logical/ExtPack/_Motion/InverterCtrl/InverterCtrl_v1/InitInverterCtrl (IEC)

#### InitInverterCtrl.st - Cyclic code
```iecst
PROGRAM _CYCLIC
	iIndexInverter := 1;
END_PROGRAM
```

### InverterGen.var
```iecst
VAR
	iIndexInverter : USINT;
END_VAR
```

### DocABB380.md
```markdown
| Doc Version | Description         | Date       | Resp       |
| ----------- | ------------------- | ---------- | ---------- |
| 1.0         | First release       | 30/10/2023 | J. Alarcón |
| 1.1         | Added state diagram | 13/11/2023 | J. Alarcón |
|             |                     |            |            |

# Related documentation

[ACS380 ABB VSD](https://efi365.sharepoint.com/:f:/r/sites/inkjet/cretaprint/oficinatecnica2/Lean%20Product%20Development/Controls/05%20Interesting%20data/ACS380%20ABB%20VSD?csf=1&web=1&e=WfV23F)

[Nice video for dummies](https://search.abb.com/library/Download.aspx?DocumentID=9AKK107492A3782&LanguageCode=en&DocumentPartId=&Action=Launch)

# How to use the package

![](.images\packageView.png)

Commands:

| Name         | Type    | Description                                 |
| ------------ | ------- | ------------------------------------------- |
| MovePositive | BOOLEAN | Starts a movement in the positive direction |
| MoveNegative | BOOLEAN | Starts a movement in the negative direction |
| Stop         | BOOLEAN | Stops the movement                          |
| Reset        | BOOLEAN | Acknowledges and quits all errors           |

Parameters:

| Name                | Type  | Description                                                                                                             |
| ------------------- | ----- | ----------------------------------------------------------------------------------------------------------------------- |
| Hardware.CpuFamilty | USINT | Used for simulation                                                                                                     |
| ControlMode         | UINT  | 0-Escalar, 1-Vectorial.                                                                                                 |
| Type                | ENUM  | INV_BR : For BR invertert                        INV_ABB : For ABB inverter                                             |
| Velocity            | INT   | Motor speed setpoint  [rpm]                                                                                             |
| DecTime             | DINT  | Time for deceleration ramp [s]. A value of 0 force the VSD to apply de max deceleration without overloading the CC bus. |
| AccTime             | DINT  | Time for acceleration ramp [s].  A value of 0 force the VSD to apply the max acceleration.                              |

ElecSignals.In:

| Name       | Type    | Description                               |
| ---------- | ------- | ----------------------------------------- |
| xBreakerOK | BOOLEAN | EFI Signal: Circuit breaker protection Ok |

Status:

| Name            | Type    | Description                                          |
| --------------- | ------- | ---------------------------------------------------- |
| Velocity        | INT     | Angular speed read from the VSD [rpm]                |
| Current         | REAL    | Motor current consumption [A]                        |
| StatusDisabled  | BOOLEAN | The inverter is switched off                         |
| StatusReady     | BOOLEAN | The motor is stopped and ready to perform a movement |
| StatusOperation | BOOLEAN | The motor is running or in quick stop                |
| StatusErrorStop | BOOLEAN | The inverter has some error                          |
| ReadyForOrders  | BOOLEAN | The inverter can receive a movement command.         |
| ErrorID         | UINT    | Error number                                         |
| ErrorText       | STRING  | Error description                                    |
| ErrorComms      | BOOLEAN | Communication error                                  |

# State diagram

Internal VSD state diagram (source EN_ACS380_FW_H_A5 doc), added in red where the package commands applies.

 ![](.images/stateDiagram.png)

# First installation configuration steps

From Factory Settings, with the PLC already loaded with the proper version:

1. VSD parameter 51.03 Set the node number

2. VSD parameter 51.02 Set the protocol profile = 1

3. VSD parameter 51.27 Refresh values. Set to 1 (it will change automatically to 0 after changes have taken effect). The communication will be stablished between the PLC and the VSD, but parameters will not be set.

4. VSD parameter 51.26 Set the force receive parameters from PLC = 1.

5. VSD parameter 51.27 Refresh values. Set to 1 (it will change automatically to 0 after changes have taken effect). After that, communication will be reseted and restablished.

6. Check that parameters have been set correctly, look inside motor parameters and check:

   1. Nominal power = 18.5 KW

   2. Nominal current = 34 A

   3. Nominal voltage = 400 V

   4. Nominal speed = 2955 rpm

   5. Nominal frequency = 50 Hz

   6. Cos fi = 0.85

7. Repeat steps 1, 2 and 3.

8. Check if VSD is already in local mode, if not, set it

9. Perform ID Run, it is a required tunning performed by the VSD whenever motor parameters are modified.

   1. Select 99.13 ID run requested, check if it is set to 3 (Standstill, no movement), if not, set it.

   2. An AFF6 Identification run warning message is shown. The panel LED starts to blink green to indicate an active warning.

   3. On the AFF6 warning, press Start to start the ID run. Do not press any control panel keys during the ID run. If you need to stop the ID run, press Stop.

   4. After the ID run is completed, the status light stops blinking. If the ID run fails, the panel shows the fault FF61 ID run

10. VSD parameter 96.07 Save parameters = 1, to save the parameters even after power off.

11. Check if VSD is already in remote mode, if not, set it.
```

### Program Logical/ExtPack/_Motion/StepperCtrl/StepperCtrl_v1/StepperX2XCtrl (IEC) - Stepper Axis X2X Control

#### StepperX2XCtrl.var
```iecst
VAR
	xInitDone : BOOL := FALSE;
	pStepperCtrl : REFERENCE TO StepperCtrlX2X_typ; (*Axis control structure (local reference to avoid doing a find & replace)*)
	oSetPosOld : INT := 0;
END_VAR
```

### Program Logical/ExtPack/_Motion/StepperCtrl/StepperCtrl_v1/InitStepperX2XCtrl (IEC) - Handling Index

#### InitStepperX2XCtrl.st - Cyclic code
```iecst
PROGRAM _CYCLIC
	(* Insert code here *)
	 gIndexStepper:= 1;
END_PROGRAM
```

### StepperCtrl.var - Global Vars
```iecst
VAR
	gIndexStepper : INT := 1;
	gAxisStepper : ARRAY[0..2] OF StepperCtrlX2X_typ;
END_VAR
```

### Program Logical/ExtPack/_Tools/EventLog/EventLog_v1/EventLogGen (IEC)

#### EventLog.var
```iecst
(********************************************************************
 * COPYRIGHT -- Bernecker + Rainer
 ********************************************************************
 * Program: EventLog
 * File: EventLog.var
 * Author: Bernecker + Rainer
 * Created: June, 2015
 ********************************************************************
 * Local variables of program EventLog
 ********************************************************************)
VAR
	EventLog : GenEventLog_typ; (*Event handling.*)
	SemFifoCreate : SemCreate; (*SemCreate Functionblock*)
	SemFifoGetInfo : SemGetInfo; (*SemGetInfo Functionblock*)
	SemIdent : UDINT;
END_VAR
```

### Library Logical/ExtPack/_Tools/EventLog/EventLog_v1/EvLogLib (IEC)

#### EventManager.st
```iecst
(* TODO: Add your comment here *)
FUNCTION_BLOCK EventManager

	//If not Semaphore, return
	IF SemId = 0 THEN
		RETURN;
	END_IF

	//Create the FIFO at init. Return while creating the FIFO
	IF NOT Init THEN
		Fifo.fCreate();
		IF Fifo.fCreate.status = ERR_OK THEN
			Fifo.fCreate.enable := FALSE;
			ident:=Fifo.fCreate.ident;
			Init:=TRUE;
		ELSIF Fifo.fCreate.status = fifoERR_FIFO_ALREADY_EXISTS THEN
			statusGetIdent:=fifoGetIdent(pFifo:= ADR('EvLog'), pIdent:=ADR(ident));
			Init:=TRUE;
		ELSIF Fifo.fCreate.status <> ERR_FUB_BUSY THEN
			Fifo.fCreate.enable := TRUE;
			Fifo.fCreate.pFifo := ADR('EvLog'); //Name of the FIFO
			Fifo.fCreate.size := 60 * SIZEOF(EventLog_typ); // XX elements size
			Fifo.fCreate.mode := fifoMODE_WRITE_UNTIL_FULL;
		END_IF
		RETURN;
	END_IF

//	//If EventLog is not configured do not execute code
//	IF ADR(EventLog)=0 THEN
//		Busy := FALSE;
//		RETURN;
//	END_IF

	//Take the information about the Stack, to review if there are item to extrack
	Fifo.fGetInfo.enable:=TRUE;
	Fifo.fGetInfo.ident := ident;
	Fifo.fGetInfo();

	IF xLoggingEvent THEN

		//Review when the Event has been logged
		IF EventLog.Event.Status = ELOG_STATUS_LOGGED THEN
			EventDataRead.Status := ELOG_STATUS_LOGGED;
			xLoggingEvent:=FALSE;

		//If the Event has not been logged, return to avoid reading another Event and crash the CPU ;-)
		ELSE
			execLogging := execLogging +1;
			RETURN;
		END_IF

	END_IF

	IF Fifo.fGetInfo.fifoUsed >0 THEN

		//Try to Acquire the Semaphore
		uiSemStatus := SemAcquire(SemId);
		IF uiSemStatus = semERR_NOT_FREE THEN
			RETURN;
		END_IF

		//Take the information about the Stack, to review if there are item to extrack
		//Read information about the Stack
		Fifo.fRead.enable := TRUE;
		Fifo.fRead.ident := ident;
		Fifo.fRead.size := SIZEOF(EventLog_typ);
		Fifo.fRead.pData := ADR(InternalEventData);
		Fifo.fRead();

		pEventData:=ADR(InternalEventData);
		EventDataRead ACCESS InternalEventData.pMyDir;
		EventDataRead.Status := ELOG_STATUS_LOGGING;

		//Text too long protection
		IF brsstrlen(ADR(EventDataRead.Text)) > 125 THEN
			brsstrcpy(ADR(EventLog.Event.AdditionalData), ADR('Text too long. Protected to avoid CPU to service'));
		ELSE
			brsstrcpy(ADR(EventLog.Event.AdditionalData), ADR(EventDataRead.Text));
		END_IF

		EventLog.Event.AdditionalDataSize := brsstrlen(ADR(EventLog.Event.AdditionalData)) + 1;
		EventLog.Event.AdditionalDataFormat := arEVENTLOG_ADDFORMAT_TEXT;

		EventLog.Event.Severity := GetSeverity(EventDataRead.Severity);
		EventLog.Event.Facility := EventDataRead.Facility;
		EventLog.Event.ErrorCode := EventDataRead.ErrorCode;

		//EventLog.Event.EnteredBy := 'TheGroup';
		GetGroupName( GenEventLog:=ADR(EventLog), EventLog:=ADR(EventDataRead));
		EventLog.Commands.WriteUserEvent:= TRUE;

		xLoggingEvent:=TRUE;

		//Release the Semaphore
		SemRelease(SemId);

		execEventData := execEventData + 1;

	END_IF

	execReview := execReview +1;

END_FUNCTION_BLOCK

FUNCTION GetGroupName

	CASE EventLog.Source OF

		ELOG_TYPE_GENERAL:
			GenEventLog.Event.EnteredBy := 'General';
		ELOG_TYPE_BAR:
			GenEventLog.Event.EnteredBy := 'Bars';
		ELOG_TYPE_BLOCK:
			GenEventLog.Event.EnteredBy := 'Blocks';
		ELOG_TYPE_SIMPLEBLOCK:
			GenEventLog.Event.EnteredBy := 'Simple Blocks';
		ELOG_TYPE_BELT:
			GenEventLog.Event.EnteredBy := 'Belt';
		ELOG_TYPE_LED:
			GenEventLog.Event.EnteredBy := 'CuringLeds';
		ELOG_TYPE_TRANS_VACUUM:
			GenEventLog.Event.EnteredBy := 'Tr. Vacuum';
		ELOG_TYPE_NONCRASH:
			GenEventLog.Event.EnteredBy := 'Non Crash';
		ELOG_TYPE_NIR:
			GenEventLog.Event.EnteredBy := 'NIR';
		ELOG_TYPE_ARCLAMP:
			GenEventLog.Event.EnteredBy := 'Arc Lamp';
		ELOG_TYPE_DETECTION:
			GenEventLog.Event.EnteredBy := 'Detection';
		ELOG_TYPE_EHD:
			GenEventLog.Event.EnteredBy := 'EHD';
		ELOG_TYPE_PAIRED_ICLA:
			GenEventLog.Event.EnteredBy := 'Pair Icla';

	END_CASE
	GetGroupName := TRUE; //Return value to avoid warning

END_FUNCTION

FUNCTION GetSeverity

	CASE Severity OF

		ELOG_SEVERITY_INFO:
			GetSeverity := arEVENTLOG_SEVERITY_INFO;
		ELOG_SEVERITY_WARNING:
			GetSeverity := arEVENTLOG_SEVERITY_WARNING;
		ELOG_SEVERITY_ERROR:
			GetSeverity := arEVENTLOG_SEVERITY_ERROR;
		ELOG_SEVERITY_SUCCESS:
			GetSeverity := arEVENTLOG_SEVERITY_SUCCESS;

	END_CASE

END_FUNCTION
```

### Program Logical/ExtPack/_Tools/SimUseRegister/SimUseRegister_1/SimUseRegister

#### FolderHandling.typ
```iecst
(********************************************************************
 * COPYRIGHT -- Bernecker + Rainer
 ********************************************************************
 * Program: FolderHandling
 * File: FolderHandling.typ
 * Author: Bernecker + Rainer
 * Created: April 17, 2009
 ********************************************************************
 * Local data types of program FolderHandling
 ********************************************************************)

TYPE
	DirHandling_Functionblock_typ : 	STRUCT
		DevLink_0 : REFERENCE TO DevLink; (*Functionblock DevLink()*)
		DirInfo_0 : DirInfo; (*Functionblock DirInfo()*)
		DirRead_0 : DirRead; (*Functionblock DirRead()*)
		DirCreate_0 : DirCreate; (*Functionblock DirCreate()*)
		DirCopy_0 : DirCopy; (*Functionblock DirCopy()*)
		DirRename_0 : DirRename; (*Functionblock DirReaname()*)
		DirDelete_0 : DirDelete; (*Functionblock DirDelete()*)
		DevMemInfo_0 : DevMemInfo; (*Functionblock DevMemInfo()*)
		GetAttributes_0 : GetAttributes; (*Functionblock GetAttributes ()*)
		SetAttributes_0 : SetAttributes; (*Functionblock SetAttributes()*)
	END_STRUCT;
	DirHandling_Data_typ : 	STRUCT
		DirName : STRING[100]; (*folder name for command bDirInfo, bDirRead, bDirCreate, bDirCopy, bDirRename, bDevMemiInfo, bGetAttributes, bSetAttributes*)
		NewDirName : STRING[100]; (*new folder name for command bdirCopy and bDirRename*)
		Device : {REDUND_UNREPLICABLE} STRING[100]; (*device name*)
		Parameter : {REDUND_UNREPLICABLE} STRING[100]; (*parameterstring for FUB DevLink()*)
		FileList : ARRAY[0..12]OF STRING[100]; (*list of files ond folders found with FUB DirRead()*)
		Step : USINT; (*step variable (255 = error step)*)
	END_STRUCT;
	DirHandling_Command_typ : 	STRUCT
		bDirRead : BOOL; (*Command: read names of file and folders*)
		bDirCreate : BOOL; (*Command: create new folder*)
		bDirRename : BOOL; (*Command: rename folder*)
		bDirCopy : BOOL; (*Command: copy a folder*)
		bDirDelete : BOOL; (*Command: delete folder*)
		bDevMemInfo : BOOL; (*Command: read information about the device*)
		bGetAttributes : BOOL; (*Command: read folder attributes*)
		bSetAttributes : BOOL; (*Command: set folder attributes*)
	END_STRUCT;
	DirHandling_typ : 	STRUCT
		Command : DirHandling_Command_typ; (*Command structure*)
		Data : DirHandling_Data_typ; (*Data structure*)
		Functionblock : DirHandling_Functionblock_typ; (*FUB structure*)
	END_STRUCT;
END_TYPE
```

#### SimUseRegister.var
```iecst
(********************************************************************
 * COPYRIGHT -- Bernecker + Rainer
 ********************************************************************
 * Program: FileHandling
 * File: FileHandling.var
 * Author: Bernecker + Rainer
 * Created: April 16, 2009
 ********************************************************************
 * Local variables of program FileHandling
 ********************************************************************)
VAR
	Handling : FileHandling_typ; (*Handlingdata for this fileio example*)
	Error : UINT; (*return value from FileIoGetSysError()*)
	FolderHandling : DirHandling_typ; (*Handlingdata for this fileio example*)
	FolderError : UINT; (*return value from FileIoGetSysError()*)
	FolderCounter : USINT; (*counter-variable for command bDirRead*)
	ReadData : fiDIR_READ_DATA; (*data-structure for command bDirRead*)
END_VAR
VAR CONSTANT
	FOLDER_SIM_REG : STRING[32] := 'SimRegister';
END_VAR
VAR
	FileNameReg : {REDUND_UNREPLICABLE} STRING[32];
	iYear : UINT;
	strYear : STRING[6];
	getTime : DTStructureGetTime;
	TimeValue : DTStructure;
	SimRegState : SimRegisterState := SIMR_STOPPED;
	FileNameAux : {REDUND_UNREPLICABLE} STRING[32];
	FileNameAuxPre : {REDUND_UNREPLICABLE} STRING[32];
	iDigits : UINT;
	xFunctionEnded : BOOL;
	xStepManaged : BOOL;
	lastHour : UINT := 99;
END_VAR
```
